LIN {X 0.308,Y -584.908,Z 581.186,A 0.000,B 0.000,C 90.000,E1 69.390} C_DIS
LIN {X -0.011,Y -580.136,Z 581.182,A 0.000,B 0.000,C 90.000,E1 68.773} C_DIS
LIN {X 0.020,Y -575.905,Z 581.179,A 0.000,B 0.000,C 90.000,E1 68.230} C_DIS
LIN {X 0.232,Y -571.249,Z 581.176,A 0.000,B 0.000,C 90.000,E1 67.667} C_DIS
LIN {X -0.295,Y -566.250,Z 581.173,A 0.000,B 0.000,C 90.000,E1 67.177} C_DIS
LIN {X 0.038,Y -560.798,Z 581.170,A 0.000,B 0.000,C 90.000,E1 66.613} C_DIS
LIN {X 0.100,Y -555.120,Z 581.167,A 0.000,B 0.000,C 90.000,E1 66.102} C_DIS
LIN {X 0.102,Y -550.770,Z 581.165,A 0.000,B 0.000,C 90.000,E1 65.741} C_DIS
LIN {X -0.055,Y -544.510,Z 581.163,A 0.000,B 0.000,C 90.000,E1 65.305} C_DIS
LIN {X 0.138,Y -539.632,Z 581.161,A 0.000,B 0.000,C 90.000,E1 64.973} C_DIS
LIN {X 0.129,Y -532.814,Z 581.159,A 0.000,B 0.000,C 90.000,E1 64.588} C_DIS
LIN {X 0.037,Y -527.787,Z 581.157,A 0.000,B 0.000,C 90.000,E1 64.332} C_DIS
LIN {X -0.007,Y -517.436,Z 581.155,A 0.000,B 0.000,C 90.000,E1 63.845} C_DIS
LIN {X -0.005,Y -503.496,Z 581.151,A 0.000,B 0.000,C 90.000,E1 63.256} C_DIS
LIN {X 0.112,Y -476.240,Z 581.145,A 0.000,B 0.000,C 90.000,E1 62.103} C_DIS
LIN {X 0.005,Y -460.881,Z 581.141,A 0.000,B 0.000,C 90.000,E1 61.435} C_DIS
LIN {X 0.181,Y -453.443,Z 581.139,A 0.000,B 0.000,C 90.000,E1 61.051} C_DIS
LIN {X 0.140,Y -453.425,Z 581.139,A 0.000,B 0.000,C 90.000,E1 61.051} C_DIS
LIN {X 0.180,Y -444.954,Z 581.117,A 0.000,B 0.000,C 90.000,E1 57.041} C_DIS
LIN {X -0.068,Y -443.758,Z 581.113,A 0.000,B 0.000,C 90.000,E1 56.421} C_DIS
LIN {X 0.017,Y -435.296,Z 581.093,A 0.000,B 0.000,C 90.000,E1 52.798} C_DIS
LIN {X 0.096,Y -437.237,Z 581.082,A 0.000,B 0.000,C 90.000,E1 50.803} C_DIS
LIN {X -0.065,Y -438.870,Z 581.073,A 0.000,B 0.000,C 90.000,E1 49.175} C_DIS
LIN {X -0.242,Y -440.515,Z 581.064,A 0.000,B 0.000,C 90.000,E1 47.553} C_DIS
LIN {X -0.085,Y -442.174,Z 581.055,A 0.000,B 0.000,C 90.000,E1 45.891} C_DIS
LIN {X -0.210,Y -443.668,Z 581.046,A 0.000,B 0.000,C 90.000,E1 44.271} C_DIS
LIN {X 0.049,Y -444.363,Z 581.040,A 0.000,B 0.000,C 90.000,E1 43.257} C_DIS
LIN {X -0.030,Y -445.165,Z 581.033,A 0.000,B 0.000,C 90.000,E1 41.962} C_DIS
LIN {X 0.265,Y -445.814,Z 581.026,A 0.000,B 0.000,C 90.000,E1 40.620} C_DIS
LIN {X -0.051,Y -446.373,Z 581.019,A 0.000,B 0.000,C 90.000,E1 39.358} C_DIS
LIN {X -0.036,Y -446.814,Z 581.010,A 0.000,B 0.000,C 90.000,E1 37.729} C_DIS
LIN {X 0.006,Y -446.976,Z 581.002,A 0.000,B 0.000,C 90.000,E1 36.423} C_DIS
LIN {X 0.148,Y -446.984,Z 580.995,A 0.000,B 0.000,C 90.000,E1 35.105} C_DIS
LIN {X -0.077,Y -446.839,Z 580.988,A 0.000,B 0.000,C 90.000,E1 33.833} C_DIS
LIN {X 0.024,Y -446.665,Z 580.975,A 0.000,B 0.000,C 90.000,E1 31.544} C_DIS
LIN {X -0.102,Y -446.477,Z 580.963,A 0.000,B 0.000,C 90.000,E1 29.283} C_DIS
LIN {X -0.067,Y -446.370,Z 580.950,A 0.000,B 0.000,C 90.000,E1 27.001} C_DIS
LIN {X -0.040,Y -446.256,Z 580.937,A 0.000,B 0.000,C 90.000,E1 24.719} C_DIS
LIN {X 0.199,Y -446.365,Z 580.930,A 0.000,B 0.000,C 90.000,E1 23.387} C_DIS
LIN {X 0.144,Y -446.539,Z 580.916,A 0.000,B 0.000,C 90.000,E1 20.791} C_DIS
LIN {X -0.247,Y -446.752,Z 580.907,A 0.000,B 0.000,C 90.000,E1 19.214} C_DIS
LIN {X 0.107,Y -447.188,Z 580.892,A 0.000,B 0.000,C 90.000,E1 16.567} C_DIS
LIN {X 0.052,Y -447.892,Z 580.880,A 0.000,B 0.000,C 90.000,E1 14.300} C_DIS
LIN {X -0.028,Y -448.946,Z 580.865,A 0.000,B 0.000,C 90.000,E1 11.715} C_DIS
LIN {X 0.196,Y -450.403,Z 580.851,A 0.000,B 0.000,C 90.000,E1 9.095} C_DIS
LIN {X 0.187,Y -451.893,Z 580.838,A 0.000,B 0.000,C 90.000,E1 6.834} C_DIS
LIN {X -0.185,Y -454.022,Z 580.824,A 0.000,B 0.000,C 90.000,E1 4.302} C_DIS
LIN {X 0.181,Y -456.138,Z 580.811,A 0.000,B 0.000,C 90.000,E1 2.007} C_DIS
LIN {X -0.091,Y -458.975,Z 580.797,A 0.000,B 0.000,C 90.000,E1 359.484} C_DIS
LIN {X 0.140,Y -462.274,Z 580.783,A 0.000,B 0.000,C 90.000,E1 356.906} C_DIS
LIN {X 0.093,Y -465.005,Z 580.772,A 0.000,B 0.000,C 90.000,E1 355.008} C_DIS
LIN {X -0.081,Y -468.314,Z 580.760,A 0.000,B 0.000,C 90.000,E1 352.818} C_DIS
LIN {X 0.216,Y -469.792,Z 580.755,A 0.000,B 0.000,C 90.000,E1 351.837} C_DIS
LIN {X -0.006,Y -472.711,Z 580.744,A 0.000,B 0.000,C 90.000,E1 349.982} C_DIS
LIN {X -0.148,Y -476.086,Z 580.732,A 0.000,B 0.000,C 90.000,E1 347.813} C_DIS
LIN {X 0.233,Y -480.226,Z 580.718,A 0.000,B 0.000,C 90.000,E1 345.283} C_DIS
LIN {X 0.061,Y -484.710,Z 580.705,A 0.000,B 0.000,C 90.000,E1 342.834} C_DIS
LIN {X 0.141,Y -488.837,Z 580.693,A 0.000,B 0.000,C 90.000,E1 340.678} C_DIS
LIN {X 0.140,Y -492.354,Z 580.683,A 0.000,B 0.000,C 90.000,E1 338.847} C_DIS
LIN {X -0.155,Y -494.607,Z 580.676,A 0.000,B 0.000,C 90.000,E1 337.667} C_DIS
LIN {X 0.039,Y -496.830,Z 580.669,A 0.000,B 0.000,C 90.000,E1 336.433} C_DIS
LIN {X 0.070,Y -499.384,Z 580.661,A 0.000,B 0.000,C 90.000,E1 334.921} C_DIS
LIN {X -0.016,Y -502.330,Z 580.651,A 0.000,B 0.000,C 90.000,E1 333.127} C_DIS
LIN {X 0.137,Y -506.065,Z 580.637,A 0.000,B 0.000,C 90.000,E1 330.717} C_DIS
LIN {X -0.120,Y -509.435,Z 580.626,A 0.000,B 0.000,C 90.000,E1 328.663} C_DIS
LIN {X -0.037,Y -512.889,Z 580.614,A 0.000,B 0.000,C 90.000,E1 326.580} C_DIS
LIN {X -0.079,Y -515.990,Z 580.605,A 0.000,B 0.000,C 90.000,E1 324.815} C_DIS
LIN {X 0.016,Y -518.630,Z 580.596,A 0.000,B 0.000,C 90.000,E1 323.336} C_DIS
LIN {X -0.084,Y -522.965,Z 580.583,A 0.000,B 0.000,C 90.000,E1 321.009} C_DIS
LIN {X 0.114,Y -529.618,Z 580.566,A 0.000,B 0.000,C 90.000,E1 317.796} C_DIS
LIN {X -0.093,Y -533.573,Z 580.558,A 0.000,B 0.000,C 90.000,E1 316.377} C_DIS
LIN {X 0.250,Y -534.789,Z 580.556,A 0.000,B 0.000,C 90.000,E1 316.053} C_DIS
LIN {X 0.019,Y -536.190,Z 580.554,A 0.000,B 0.000,C 90.000,E1 315.648} C_DIS
LIN {X 0.026,Y -537.834,Z 580.552,A 0.000,B 0.000,C 90.000,E1 315.324} C_DIS
LIN {X -0.189,Y -540.578,Z 580.549,A 0.000,B 0.000,C 90.000,E1 314.919} C_DIS
LIN {X 0.043,Y -544.352,Z 580.547,A 0.000,B 0.000,C 90.000,E1 314.433} C_DIS
LIN {X -0.320,Y -548.922,Z 580.544,A 0.000,B 0.000,C 90.000,E1 314.028} C_DIS
LIN {X 0.000,Y -553.189,Z 580.542,A 0.000,B 0.000,C 90.000,E1 313.623} C_DIS
LIN {X 0.089,Y -558.609,Z 580.540,A 0.000,B 0.000,C 90.000,E1 313.176} C_DIS
LIN {X 0.161,Y -572.961,Z 580.534,A 0.000,B 0.000,C 90.000,E1 312.123} C_DIS
LIN {X -0.240,Y -592.219,Z 580.526,A 0.000,B 0.000,C 90.000,E1 310.782} C_DIS
LIN {X -0.096,Y -597.922,Z 580.524,A 0.000,B 0.000,C 90.000,E1 310.334} C_DIS
LIN {X -0.088,Y -604.769,Z 580.521,A 0.000,B 0.000,C 90.000,E1 309.769} C_DIS
LIN {X -0.314,Y -611.213,Z 580.518,A 0.000,B 0.000,C 90.000,E1 309.197} C_DIS
LIN {X 0.067,Y -616.222,Z 580.515,A 0.000,B 0.000,C 90.000,E1 308.669} C_DIS
LIN {X -0.076,Y -620.961,Z 580.512,A 0.000,B 0.000,C 90.000,E1 308.177} C_DIS
LIN {X -0.260,Y -624.426,Z 580.510,A 0.000,B 0.000,C 90.000,E1 307.810} C_DIS
LIN {X -0.030,Y -632.937,Z 580.504,A 0.000,B 0.000,C 90.000,E1 306.790} C_DIS
LIN {X -0.173,Y -636.872,Z 580.502,A 0.000,B 0.000,C 90.000,E1 306.297} C_DIS
LIN {X 0.125,Y -643.552,Z 580.497,A 0.000,B 0.000,C 90.000,E1 305.391} C_DIS
LIN {X 0.042,Y -648.595,Z 580.493,A 0.000,B 0.000,C 90.000,E1 304.659} C_DIS
LIN {X -0.175,Y -650.918,Z 580.491,A 0.000,B 0.000,C 90.000,E1 304.326} C_DIS
LIN {X -0.109,Y -654.518,Z 580.487,A 0.000,B 0.000,C 90.000,E1 303.706} C_DIS
LIN {X -0.015,Y -658.416,Z 580.483,A 0.000,B 0.000,C 90.000,E1 302.959} C_DIS
LIN {X 0.058,Y -661.330,Z 580.480,A 0.000,B 0.000,C 90.000,E1 302.339} C_DIS
LIN {X 0.213,Y -664.599,Z 580.476,A 0.000,B 0.000,C 90.000,E1 301.592} C_DIS
LIN {X 0.119,Y -669.758,Z 580.469,A 0.000,B 0.000,C 90.000,E1 300.384} C_DIS
LIN {X 0.016,Y -672.719,Z 580.465,A 0.000,B 0.000,C 90.000,E1 299.667} C_DIS
LIN {X -0.056,Y -675.468,Z 580.461,A 0.000,B 0.000,C 90.000,E1 298.949} C_DIS
LIN {X -0.100,Y -677.959,Z 580.457,A 0.000,B 0.000,C 90.000,E1 298.231} C_DIS
LIN {X 0.279,Y -681.824,Z 580.450,A 0.000,B 0.000,C 90.000,E1 297.001} C_DIS
LIN {X 0.081,Y -683.228,Z 580.448,A 0.000,B 0.000,C 90.000,E1 296.539} C_DIS
LIN {X -0.201,Y -684.258,Z 580.444,A 0.000,B 0.000,C 90.000,E1 295.848} C_DIS
LIN {X 0.013,Y -683.895,Z 580.442,A 0.000,B 0.000,C 90.000,E1 295.591} C_DIS
LIN {X 0.150,Y -682.857,Z 580.440,A 0.000,B 0.000,C 90.000,E1 295.103} C_DIS
LIN {X -0.363,Y -682.292,Z 580.439,A 0.000,B 0.000,C 90.000,E1 295.027} C_DIS
LIN {X -0.256,Y -681.396,Z 580.438,A 0.000,B 0.000,C 90.000,E1 294.899} C_DIS
LIN {X 0.149,Y -677.002,Z 580.436,A 0.000,B 0.000,C 90.000,E1 294.387} C_DIS
LIN {X 0.244,Y -675.191,Z 580.435,A 0.000,B 0.000,C 90.000,E1 294.259} C_DIS
LIN {X -0.231,Y -669.405,Z 580.433,A 0.000,B 0.000,C 90.000,E1 294.027} C_DIS
LIN {X 0.155,Y -667.577,Z 580.433,A 0.000,B 0.000,C 90.000,E1 293.898} C_DIS
LIN {X 0.000,Y -660.359,Z 580.432,A 0.000,B 0.000,C 90.000,E1 293.695} C_DIS
LIN {X -0.005,Y -658.269,Z 580.431,A 0.000,B 0.000,C 90.000,E1 293.643} C_DIS
LIN {X 0.273,Y -632.150,Z 580.428,A 0.000,B 0.000,C 90.000,E1 293.078} C_DIS
LIN {X -0.006,Y -618.722,Z 580.427,A 0.000,B 0.000,C 90.000,E1 292.770} C_DIS
LIN {X 0.232,Y -598.679,Z 580.423,A 0.000,B 0.000,C 90.000,E1 292.153} C_DIS
LIN {X -0.237,Y -572.595,Z 580.419,A 0.000,B 0.000,C 90.000,E1 291.354} C_DIS
LIN {X 0.149,Y -566.186,Z 580.417,A 0.000,B 0.000,C 90.000,E1 291.046} C_DIS
LIN {X -0.102,Y -562.883,Z 580.416,A 0.000,B 0.000,C 90.000,E1 290.844} C_DIS
LIN {X -0.133,Y -562.840,Z 580.416,A 0.000,B 0.000,C 90.000,E1 290.844} C_DIS
LIN {X -0.190,Y -561.903,Z 580.415,A 0.000,B 0.000,C 90.000,E1 290.663} C_DIS
LIN {X -0.175,Y -561.379,Z 580.412,A 0.000,B 0.000,C 90.000,E1 290.248} C_DIS
LIN {X -0.231,Y -561.567,Z 580.405,A 0.000,B 0.000,C 90.000,E1 288.960} C_DIS
LIN {X -0.279,Y -561.238,Z 580.398,A 0.000,B 0.000,C 90.000,E1 287.583} C_DIS
LIN {X -0.069,Y -560.943,Z 580.393,A 0.000,B 0.000,C 90.000,E1 286.732} C_DIS
LIN {X 0.114,Y -560.513,Z 580.387,A 0.000,B 0.000,C 90.000,E1 285.607} C_DIS
LIN {X -0.101,Y -559.747,Z 580.379,A 0.000,B 0.000,C 90.000,E1 284.245} C_DIS
LIN {X 0.212,Y -558.948,Z 580.371,A 0.000,B 0.000,C 90.000,E1 282.827} C_DIS
LIN {X -0.020,Y -558.032,Z 580.362,A 0.000,B 0.000,C 90.000,E1 281.186} C_DIS
LIN {X 0.173,Y -557.035,Z 580.353,A 0.000,B 0.000,C 90.000,E1 279.500} C_DIS
LIN {X -0.158,Y -556.088,Z 580.342,A 0.000,B 0.000,C 90.000,E1 277.587} C_DIS
LIN {X -0.217,Y -555.447,Z 580.334,A 0.000,B 0.000,C 90.000,E1 276.201} C_DIS
LIN {X 0.007,Y -554.575,Z 580.320,A 0.000,B 0.000,C 90.000,E1 273.669} C_DIS
LIN {X -0.014,Y -554.033,Z 580.310,A 0.000,B 0.000,C 90.000,E1 271.718} C_DIS
LIN {X -0.149,Y -553.451,Z 580.300,A 0.000,B 0.000,C 90.000,E1 270.057} C_DIS
LIN {X 0.189,Y -552.885,Z 580.293,A 0.000,B 0.000,C 90.000,E1 268.625} C_DIS
LIN {X 0.129,Y -552.074,Z 580.282,A 0.000,B 0.000,C 90.000,E1 266.674} C_DIS
LIN {X -0.101,Y -551.405,Z 580.274,A 0.000,B 0.000,C 90.000,E1 265.298} C_DIS
LIN {X -0.251,Y -550.616,Z 580.266,A 0.000,B 0.000,C 90.000,E1 263.913} C_DIS
LIN {X 0.037,Y -549.903,Z 580.260,A 0.000,B 0.000,C 90.000,E1 262.761} C_DIS
LIN {X 0.277,Y -549.162,Z 580.255,A 0.000,B 0.000,C 90.000,E1 261.894} C_DIS
LIN {X 0.171,Y -547.801,Z 580.247,A 0.000,B 0.000,C 90.000,E1 260.500} C_DIS
LIN {X -0.109,Y -545.300,Z 580.233,A 0.000,B 0.000,C 90.000,E1 257.993} C_DIS
LIN {X 0.028,Y -543.540,Z 580.224,A 0.000,B 0.000,C 90.000,E1 256.284} C_DIS
LIN {X 0.123,Y -541.724,Z 580.214,A 0.000,B 0.000,C 90.000,E1 254.574} C_DIS
LIN {X 0.028,Y -540.537,Z 580.208,A 0.000,B 0.000,C 90.000,E1 253.449} C_DIS
LIN {X 0.067,Y -539.198,Z 580.202,A 0.000,B 0.000,C 90.000,E1 252.308} C_DIS
LIN {X 0.085,Y -537.687,Z 580.195,A 0.000,B 0.000,C 90.000,E1 251.167} C_DIS
LIN {X -0.039,Y -535.497,Z 580.188,A 0.000,B 0.000,C 90.000,E1 249.752} C_DIS
LIN {X 0.103,Y -533.530,Z 580.181,A 0.000,B 0.000,C 90.000,E1 248.592} C_DIS
LIN {X 0.214,Y -531.881,Z 580.176,A 0.000,B 0.000,C 90.000,E1 247.720} C_DIS
LIN {X -0.011,Y -528.945,Z 580.168,A 0.000,B 0.000,C 90.000,E1 246.305} C_DIS
LIN {X 0.133,Y -525.899,Z 580.160,A 0.000,B 0.000,C 90.000,E1 244.845} C_DIS
LIN {X 0.224,Y -522.723,Z 580.152,A 0.000,B 0.000,C 90.000,E1 243.384} C_DIS
LIN {X 0.111,Y -520.028,Z 580.146,A 0.000,B 0.000,C 90.000,E1 242.231} C_DIS
LIN {X 0.201,Y -517.136,Z 580.139,A 0.000,B 0.000,C 90.000,E1 241.051} C_DIS
LIN {X -0.111,Y -514.849,Z 580.134,A 0.000,B 0.000,C 90.000,E1 240.205} C_DIS
LIN {X 0.161,Y -511.634,Z 580.128,A 0.000,B 0.000,C 90.000,E1 238.997} C_DIS
LIN {X 0.014,Y -507.672,Z 580.120,A 0.000,B 0.000,C 90.000,E1 237.533} C_DIS
LIN {X 0.132,Y -505.254,Z 580.115,A 0.000,B 0.000,C 90.000,E1 236.628} C_DIS
LIN {X -0.284,Y -501.072,Z 580.106,A 0.000,B 0.000,C 90.000,E1 235.182} C_DIS
LIN {X 0.070,Y -491.975,Z 580.088,A 0.000,B 0.000,C 90.000,E1 231.823} C_DIS
LIN {X 0.100,Y -485.568,Z 580.074,A 0.000,B 0.000,C 90.000,E1 229.380} C_DIS
LIN {X -0.122,Y -479.269,Z 580.061,A 0.000,B 0.000,C 90.000,E1 226.944} C_DIS
LIN {X -0.107,Y -474.704,Z 580.050,A 0.000,B 0.000,C 90.000,E1 225.081} C_DIS
LIN {X 0.061,Y -471.030,Z 580.042,A 0.000,B 0.000,C 90.000,E1 223.500} C_DIS
LIN {X 0.227,Y -466.705,Z 580.031,A 0.000,B 0.000,C 90.000,E1 221.595} C_DIS
LIN {X 0.063,Y -461.888,Z 580.019,A 0.000,B 0.000,C 90.000,E1 219.402} C_DIS
LIN {X -0.183,Y -457.842,Z 580.008,A 0.000,B 0.000,C 90.000,E1 217.523} C_DIS
LIN {X 0.029,Y -455.160,Z 580.001,A 0.000,B 0.000,C 90.000,E1 216.217} C_DIS
LIN {X 0.102,Y -451.223,Z 579.991,A 0.000,B 0.000,C 90.000,E1 214.278} C_DIS
LIN {X 0.088,Y -447.488,Z 579.980,A 0.000,B 0.000,C 90.000,E1 212.339} C_DIS
LIN {X -0.051,Y -443.386,Z 579.967,A 0.000,B 0.000,C 90.000,E1 210.079} C_DIS
LIN {X 0.042,Y -439.856,Z 579.956,A 0.000,B 0.000,C 90.000,E1 208.103} C_DIS
LIN {X -0.190,Y -436.993,Z 579.947,A 0.000,B 0.000,C 90.000,E1 206.488} C_DIS
LIN {X 0.127,Y -433.611,Z 579.936,A 0.000,B 0.000,C 90.000,E1 204.463} C_DIS
LIN {X 0.183,Y -430.314,Z 579.925,A 0.000,B 0.000,C 90.000,E1 202.461} C_DIS
LIN {X -0.008,Y -427.234,Z 579.914,A 0.000,B 0.000,C 90.000,E1 200.482} C_DIS
LIN {X -0.029,Y -424.300,Z 579.903,A 0.000,B 0.000,C 90.000,E1 198.471} C_DIS
LIN {X 0.019,Y -421.538,Z 579.891,A 0.000,B 0.000,C 90.000,E1 196.441} C_DIS
LIN {X -0.160,Y -419.418,Z 579.882,A 0.000,B 0.000,C 90.000,E1 194.773} C_DIS
LIN {X -0.082,Y -417.143,Z 579.873,A 0.000,B 0.000,C 90.000,E1 193.063} C_DIS
LIN {X 0.117,Y -412.756,Z 579.855,A 0.000,B 0.000,C 90.000,E1 189.962} C_DIS
LIN {X -0.078,Y -409.511,Z 579.840,A 0.000,B 0.000,C 90.000,E1 187.239} C_DIS
LIN {X -0.053,Y -407.085,Z 579.829,A 0.000,B 0.000,C 90.000,E1 185.163} C_DIS
LIN {X 0.132,Y -403.146,Z 579.807,A 0.000,B 0.000,C 90.000,E1 181.318} C_DIS
LIN {X -0.164,Y -401.108,Z 579.792,A 0.000,B 0.000,C 90.000,E1 178.568} C_DIS
LIN {X -0.157,Y -399.309,Z 579.773,A 0.000,B 0.000,C 90.000,E1 175.065} C_DIS
LIN {X -0.033,Y -398.643,Z 579.759,A 0.000,B 0.000,C 90.000,E1 172.591} C_DIS
LIN {X 0.181,Y -398.286,Z 579.741,A 0.000,B 0.000,C 90.000,E1 169.398} C_DIS
LIN {X -0.180,Y -398.631,Z 579.722,A 0.000,B 0.000,C 90.000,E1 165.936} C_DIS
LIN {X 0.023,Y -399.249,Z 579.708,A 0.000,B 0.000,C 90.000,E1 163.449} C_DIS
LIN {X -0.083,Y -400.233,Z 579.693,A 0.000,B 0.000,C 90.000,E1 160.659} C_DIS
LIN {X 0.048,Y -401.182,Z 579.681,A 0.000,B 0.000,C 90.000,E1 158.539} C_DIS
LIN {X 0.061,Y -402.511,Z 579.665,A 0.000,B 0.000,C 90.000,E1 155.741} C_DIS
LIN {X 0.154,Y -403.230,Z 579.658,A 0.000,B 0.000,C 90.000,E1 154.332} C_DIS
LIN {X -0.023,Y -404.157,Z 579.648,A 0.000,B 0.000,C 90.000,E1 152.615} C_DIS
LIN {X -0.067,Y -404.840,Z 579.640,A 0.000,B 0.000,C 90.000,E1 151.229} C_DIS
LIN {X 0.165,Y -405.618,Z 579.630,A 0.000,B 0.000,C 90.000,E1 149.459} C_DIS
LIN {X 0.142,Y -406.155,Z 579.623,A 0.000,B 0.000,C 90.000,E1 148.074} C_DIS
LIN {X 0.034,Y -406.709,Z 579.611,A 0.000,B 0.000,C 90.000,E1 146.008} C_DIS
LIN {X 0.031,Y -407.099,Z 579.602,A 0.000,B 0.000,C 90.000,E1 144.276} C_DIS
LIN {X -0.060,Y -407.438,Z 579.592,A 0.000,B 0.000,C 90.000,E1 142.557} C_DIS
LIN {X 0.105,Y -407.734,Z 579.582,A 0.000,B 0.000,C 90.000,E1 140.803} C_DIS
LIN {X -0.203,Y -408.076,Z 579.571,A 0.000,B 0.000,C 90.000,E1 138.771} C_DIS
LIN {X -0.226,Y -408.318,Z 579.563,A 0.000,B 0.000,C 90.000,E1 137.391} C_DIS
LIN {X -0.005,Y -408.510,Z 579.548,A 0.000,B 0.000,C 90.000,E1 134.595} C_DIS
LIN {X 0.105,Y -408.746,Z 579.538,A 0.000,B 0.000,C 90.000,E1 132.852} C_DIS
LIN {X -0.061,Y -408.923,Z 579.529,A 0.000,B 0.000,C 90.000,E1 131.148} C_DIS
LIN {X -0.075,Y -408.865,Z 579.521,A 0.000,B 0.000,C 90.000,E1 129.769} C_DIS
LIN {X -0.027,Y -408.644,Z 579.513,A 0.000,B 0.000,C 90.000,E1 128.338} C_DIS
LIN {X 0.019,Y -415.544,Z 579.500,A 0.000,B 0.000,C 90.000,E1 125.964} C_DIS
LIN {X 0.103,Y -425.936,Z 579.477,A 0.000,B 0.000,C 90.000,E1 121.878} C_DIS
LIN {X 0.056,Y -430.944,Z 579.468,A 0.000,B 0.000,C 90.000,E1 120.207} C_DIS
LIN {X 0.025,Y -432.452,Z 579.464,A 0.000,B 0.000,C 90.000,E1 119.539} C_DIS
LIN {X -0.014,Y -432.527,Z 579.464,A 0.000,B 0.000,C 90.000,E1 119.539} C_DIS
LIN {X 0.020,Y -450.020,Z 579.460,A 0.000,B 0.000,C 90.000,E1 118.743} C_DIS
LIN {X 0.056,Y -470.512,Z 579.454,A 0.000,B 0.000,C 90.000,E1 117.769} C_DIS
LIN {X -0.135,Y -482.285,Z 579.451,A 0.000,B 0.000,C 90.000,E1 117.206} C_DIS
LIN {X -0.248,Y -488.933,Z 579.449,A 0.000,B 0.000,C 90.000,E1 116.873} C_DIS
LIN {X 0.252,Y -497.099,Z 579.447,A 0.000,B 0.000,C 90.000,E1 116.360} C_DIS
LIN {X 0.075,Y -508.510,Z 579.443,A 0.000,B 0.000,C 90.000,E1 115.720} C_DIS
LIN {X 0.263,Y -516.409,Z 579.440,A 0.000,B 0.000,C 90.000,E1 115.207} C_DIS
LIN {X 0.035,Y -522.640,Z 579.438,A 0.000,B 0.000,C 90.000,E1 114.823} C_DIS
LIN {X -0.331,Y -530.462,Z 579.435,A 0.000,B 0.000,C 90.000,E1 114.335} C_DIS
LIN {X -0.211,Y -537.899,Z 579.432,A 0.000,B 0.000,C 90.000,E1 113.770} C_DIS
LIN {X 0.206,Y -542.356,Z 579.430,A 0.000,B 0.000,C 90.000,E1 113.387} C_DIS
LIN {X -0.102,Y -548.016,Z 579.427,A 0.000,B 0.000,C 90.000,E1 112.950} C_DIS
LIN {X -0.113,Y -552.213,Z 579.425,A 0.000,B 0.000,C 90.000,E1 112.589} C_DIS
LIN {X -0.037,Y -557.502,Z 579.423,A 0.000,B 0.000,C 90.000,E1 112.078} C_DIS
LIN {X 0.017,Y -562.507,Z 579.420,A 0.000,B 0.000,C 90.000,E1 111.535} C_DIS
LIN {X 0.232,Y -565.857,Z 579.417,A 0.000,B 0.000,C 90.000,E1 111.099} C_DIS
LIN {X 0.130,Y -567.039,Z 579.417,A 0.000,B 0.000,C 90.000,E1 110.972} C_DIS
LIN {X 0.169,Y -569.961,Z 579.414,A 0.000,B 0.000,C 90.000,E1 110.556} C_DIS
LIN {X -0.020,Y -571.984,Z 579.413,A 0.000,B 0.000,C 90.000,E1 110.301} C_DIS
LIN {X 0.047,Y -574.436,Z 579.411,A 0.000,B 0.000,C 90.000,E1 109.885} C_DIS
LIN {X -0.311,Y -577.683,Z 579.408,A 0.000,B 0.000,C 90.000,E1 109.396} C_DIS
LIN {X -0.102,Y -580.786,Z 579.405,A 0.000,B 0.000,C 90.000,E1 108.833} C_DIS
LIN {X 0.154,Y -584.940,Z 579.400,A 0.000,B 0.000,C 90.000,E1 108.000} C_DIS
LIN {X -0.097,Y -588.746,Z 579.396,A 0.000,B 0.000,C 90.000,E1 107.221} C_DIS
LIN {X -0.312,Y -592.321,Z 579.391,A 0.000,B 0.000,C 90.000,E1 106.441} C_DIS
LIN {X -0.226,Y -596.739,Z 579.385,A 0.000,B 0.000,C 90.000,E1 105.371} C_DIS
LIN {X -0.082,Y -598.762,Z 579.382,A 0.000,B 0.000,C 90.000,E1 104.828} C_DIS
LIN {X -0.058,Y -602.657,Z 579.377,A 0.000,B 0.000,C 90.000,E1 103.772} C_DIS
LIN {X -0.169,Y -609.216,Z 579.366,A 0.000,B 0.000,C 90.000,E1 101.951} C_DIS
LIN {X 0.108,Y -614.874,Z 579.358,A 0.000,B 0.000,C 90.000,E1 100.366} C_DIS
LIN {X 0.242,Y -618.538,Z 579.352,A 0.000,B 0.000,C 90.000,E1 99.321} C_DIS
LIN {X -0.280,Y -622.050,Z 579.346,A 0.000,B 0.000,C 90.000,E1 98.341} C_DIS
LIN {X -0.049,Y -625.451,Z 579.341,A 0.000,B 0.000,C 90.000,E1 97.296} C_DIS
LIN {X 0.146,Y -628.687,Z 579.335,A 0.000,B 0.000,C 90.000,E1 96.258} C_DIS
LIN {X -0.022,Y -630.938,Z 579.331,A 0.000,B 0.000,C 90.000,E1 95.511} C_DIS
LIN {X -0.112,Y -633.026,Z 579.326,A 0.000,B 0.000,C 90.000,E1 94.759} C_DIS
LIN {X 0.129,Y -635.367,Z 579.321,A 0.000,B 0.000,C 90.000,E1 93.726} C_DIS
LIN {X 0.024,Y -636.872,Z 579.317,A 0.000,B 0.000,C 90.000,E1 92.980} C_DIS
LIN {X -0.096,Y -638.283,Z 579.312,A 0.000,B 0.000,C 90.000,E1 92.236} C_DIS
LIN {X -0.178,Y -639.470,Z 579.308,A 0.000,B 0.000,C 90.000,E1 91.489} C_DIS
LIN {X 0.133,Y -640.660,Z 579.303,A 0.000,B 0.000,C 90.000,E1 90.458} C_DIS
LIN {X 0.059,Y -641.301,Z 579.298,A 0.000,B 0.000,C 90.000,E1 89.714} C_DIS
LIN {X -0.009,Y -641.704,Z 579.294,A 0.000,B 0.000,C 90.000,E1 88.969} C_DIS
LIN {X -0.079,Y -641.787,Z 579.290,A 0.000,B 0.000,C 90.000,E1 88.224} C_DIS
LIN {X 0.278,Y -641.521,Z 579.285,A 0.000,B 0.000,C 90.000,E1 87.192} C_DIS
LIN {X 0.234,Y -641.094,Z 579.280,A 0.000,B 0.000,C 90.000,E1 86.445} C_DIS
LIN {X -0.056,Y -640.223,Z 579.275,A 0.000,B 0.000,C 90.000,E1 85.469} C_DIS
LIN {X 0.333,Y -639.053,Z 579.269,A 0.000,B 0.000,C 90.000,E1 84.432} C_DIS
LIN {X -0.111,Y -638.402,Z 579.266,A 0.000,B 0.000,C 90.000,E1 83.970} C_DIS
LIN {X 0.259,Y -636.795,Z 579.261,A 0.000,B 0.000,C 90.000,E1 82.932} C_DIS
LIN {X 0.160,Y -635.277,Z 579.257,A 0.000,B 0.000,C 90.000,E1 82.186} C_DIS
LIN {X -0.062,Y -633.032,Z 579.251,A 0.000,B 0.000,C 90.000,E1 81.197} C_DIS
LIN {X -0.112,Y -631.199,Z 579.247,A 0.000,B 0.000,C 90.000,E1 80.443} C_DIS
LIN {X 0.236,Y -628.482,Z 579.241,A 0.000,B 0.000,C 90.000,E1 79.398} C_DIS
LIN {X -0.073,Y -625.599,Z 579.236,A 0.000,B 0.000,C 90.000,E1 78.409} C_DIS
LIN {X -0.295,Y -622.502,Z 579.230,A 0.000,B 0.000,C 90.000,E1 77.409} C_DIS
LIN {X 0.270,Y -619.915,Z 579.226,A 0.000,B 0.000,C 90.000,E1 76.589} C_DIS
LIN {X 0.201,Y -617.142,Z 579.221,A 0.000,B 0.000,C 90.000,E1 75.825} C_DIS
LIN {X 0.259,Y -614.243,Z 579.217,A 0.000,B 0.000,C 90.000,E1 75.046} C_DIS
LIN {X 0.128,Y -611.065,Z 579.213,A 0.000,B 0.000,C 90.000,E1 74.283} C_DIS
LIN {X 0.130,Y -607.605,Z 579.208,A 0.000,B 0.000,C 90.000,E1 73.504} C_DIS
LIN {X 0.050,Y -603.190,Z 579.203,A 0.000,B 0.000,C 90.000,E1 72.598} C_DIS
LIN {X -0.073,Y -597.683,Z 579.198,A 0.000,B 0.000,C 90.000,E1 71.583} C_DIS
LIN {X 0.101,Y -593.982,Z 579.194,A 0.000,B 0.000,C 90.000,E1 70.913} C_DIS
LIN {X 0.221,Y -588.281,Z 579.189,A 0.000,B 0.000,C 90.000,E1 70.007} C_DIS
LIN {X -0.236,Y -584.628,Z 579.186,A 0.000,B 0.000,C 90.000,E1 69.518} C_DIS
LIN {X 0.037,Y -580.649,Z 579.183,A 0.000,B 0.000,C 90.000,E1 68.954} C_DIS
LIN {X -0.131,Y -575.504,Z 579.180,A 0.000,B 0.000,C 90.000,E1 68.337} C_DIS
LIN {X 0.265,Y -571.069,Z 579.177,A 0.000,B 0.000,C 90.000,E1 67.794} C_DIS
LIN {X 0.104,Y -565.017,Z 579.173,A 0.000,B 0.000,C 90.000,E1 67.177} C_DIS
LIN {X 0.309,Y -561.269,Z 579.171,A 0.000,B 0.000,C 90.000,E1 66.794} C_DIS
LIN {X 0.031,Y -556.038,Z 579.169,A 0.000,B 0.000,C 90.000,E1 66.357} C_DIS
LIN {X -0.113,Y -550.476,Z 579.166,A 0.000,B 0.000,C 90.000,E1 65.921} C_DIS
LIN {X -0.272,Y -544.106,Z 579.164,A 0.000,B 0.000,C 90.000,E1 65.485} C_DIS
LIN {X -0.084,Y -539.070,Z 579.162,A 0.000,B 0.000,C 90.000,E1 65.153} C_DIS
LIN {X -0.184,Y -532.318,Z 579.160,A 0.000,B 0.000,C 90.000,E1 64.793} C_DIS
LIN {X -0.242,Y -527.296,Z 579.158,A 0.000,B 0.000,C 90.000,E1 64.537} C_DIS
LIN {X -0.051,Y -516.811,Z 579.156,A 0.000,B 0.000,C 90.000,E1 64.024} C_DIS
LIN {X -0.108,Y -501.135,Z 579.152,A 0.000,B 0.000,C 90.000,E1 63.384} C_DIS
LIN {X 0.003,Y -471.916,Z 579.145,A 0.000,B 0.000,C 90.000,E1 62.153} C_DIS
LIN {X -0.103,Y -458.508,Z 579.142,A 0.000,B 0.000,C 90.000,E1 61.563} C_DIS
LIN {X 0.267,Y -454.174,Z 579.141,A 0.000,B 0.000,C 90.000,E1 61.307} C_DIS
LIN {X 0.226,Y -454.082,Z 579.141,A 0.000,B 0.000,C 90.000,E1 61.307} C_DIS
LIN {X 0.113,Y -445.458,Z 579.119,A 0.000,B 0.000,C 90.000,E1 57.327} C_DIS
LIN {X -0.076,Y -443.629,Z 579.113,A 0.000,B 0.000,C 90.000,E1 56.373} C_DIS
LIN {X 0.064,Y -435.664,Z 579.094,A 0.000,B 0.000,C 90.000,E1 52.970} C_DIS
LIN {X -0.269,Y -437.926,Z 579.082,A 0.000,B 0.000,C 90.000,E1 50.803} C_DIS
LIN {X -0.131,Y -439.606,Z 579.073,A 0.000,B 0.000,C 90.000,E1 49.138} C_DIS
LIN {X 0.041,Y -441.307,Z 579.064,A 0.000,B 0.000,C 90.000,E1 47.472} C_DIS
LIN {X 0.216,Y -442.997,Z 579.055,A 0.000,B 0.000,C 90.000,E1 45.810} C_DIS
LIN {X 0.127,Y -444.205,Z 579.047,A 0.000,B 0.000,C 90.000,E1 44.514} C_DIS
LIN {X 0.071,Y -444.992,Z 579.042,A 0.000,B 0.000,C 90.000,E1 43.542} C_DIS
LIN {X 0.029,Y -445.822,Z 579.035,A 0.000,B 0.000,C 90.000,E1 42.243} C_DIS
LIN {X 0.006,Y -446.496,Z 579.028,A 0.000,B 0.000,C 90.000,E1 40.943} C_DIS
LIN {X -0.011,Y -447.051,Z 579.020,A 0.000,B 0.000,C 90.000,E1 39.644} C_DIS
LIN {X 0.040,Y -447.436,Z 579.013,A 0.000,B 0.000,C 90.000,E1 38.338} C_DIS
LIN {X 0.100,Y -447.659,Z 579.006,A 0.000,B 0.000,C 90.000,E1 37.030} C_DIS
LIN {X 0.157,Y -447.733,Z 578.999,A 0.000,B 0.000,C 90.000,E1 35.724} C_DIS
LIN {X 0.011,Y -447.546,Z 578.990,A 0.000,B 0.000,C 90.000,E1 34.119} C_DIS
LIN {X -0.245,Y -447.280,Z 578.977,A 0.000,B 0.000,C 90.000,E1 31.878} C_DIS
LIN {X 0.185,Y -447.085,Z 578.966,A 0.000,B 0.000,C 90.000,E1 29.873} C_DIS
LIN {X -0.146,Y -446.992,Z 578.959,A 0.000,B 0.000,C 90.000,E1 28.615} C_DIS
LIN {X -0.233,Y -446.874,Z 578.950,A 0.000,B 0.000,C 90.000,E1 27.001} C_DIS
LIN {X -0.060,Y -446.713,Z 578.939,A 0.000,B 0.000,C 90.000,E1 25.027} C_DIS
LIN {X 0.054,Y -446.776,Z 578.930,A 0.000,B 0.000,C 90.000,E1 23.387} C_DIS
LIN {X 0.141,Y -446.925,Z 578.917,A 0.000,B 0.000,C 90.000,E1 21.099} C_DIS
LIN {X 0.196,Y -447.102,Z 578.907,A 0.000,B 0.000,C 90.000,E1 19.141} C_DIS
LIN {X -0.007,Y -447.486,Z 578.892,A 0.000,B 0.000,C 90.000,E1 16.567} C_DIS
LIN {X -0.054,Y -448.174,Z 578.879,A 0.000,B 0.000,C 90.000,E1 14.300} C_DIS
LIN {X -0.126,Y -449.216,Z 578.865,A 0.000,B 0.000,C 90.000,E1 11.715} C_DIS
LIN {X -0.142,Y -450.845,Z 578.849,A 0.000,B 0.000,C 90.000,E1 8.803} C_DIS
LIN {X -0.147,Y -452.348,Z 578.836,A 0.000,B 0.000,C 90.000,E1 6.543} C_DIS
LIN {X -0.064,Y -454.495,Z 578.822,A 0.000,B 0.000,C 90.000,E1 3.955} C_DIS
LIN {X -0.153,Y -456.621,Z 578.810,A 0.000,B 0.000,C 90.000,E1 1.718} C_DIS
LIN {X -0.090,Y -459.111,Z 578.797,A 0.000,B 0.000,C 90.000,E1 359.484} C_DIS
LIN {X 0.144,Y -462.399,Z 578.783,A 0.000,B 0.000,C 90.000,E1 356.906} C_DIS
LIN {X 0.101,Y -465.118,Z 578.772,A 0.000,B 0.000,C 90.000,E1 355.008} C_DIS
LIN {X -0.071,Y -468.411,Z 578.760,A 0.000,B 0.000,C 90.000,E1 352.818} C_DIS
LIN {X 0.228,Y -469.885,Z 578.755,A 0.000,B 0.000,C 90.000,E1 351.837} C_DIS
LIN {X 0.008,Y -472.795,Z 578.744,A 0.000,B 0.000,C 90.000,E1 349.982} C_DIS
LIN {X -0.131,Y -476.160,Z 578.732,A 0.000,B 0.000,C 90.000,E1 347.813} C_DIS
LIN {X 0.101,Y -480.818,Z 578.717,A 0.000,B 0.000,C 90.000,E1 344.991} C_DIS
LIN {X -0.063,Y -484.724,Z 578.705,A 0.000,B 0.000,C 90.000,E1 342.851} C_DIS
LIN {X 0.161,Y -488.870,Z 578.693,A 0.000,B 0.000,C 90.000,E1 340.678} C_DIS
LIN {X 0.161,Y -492.383,Z 578.683,A 0.000,B 0.000,C 90.000,E1 338.847} C_DIS
LIN {X -0.134,Y -494.669,Z 578.676,A 0.000,B 0.000,C 90.000,E1 337.667} C_DIS
LIN {X 0.114,Y -497.400,Z 578.667,A 0.000,B 0.000,C 90.000,E1 336.125} C_DIS
LIN {X -0.299,Y -499.940,Z 578.659,A 0.000,B 0.000,C 90.000,E1 334.665} C_DIS
LIN {X 0.009,Y -502.421,Z 578.651,A 0.000,B 0.000,C 90.000,E1 333.127} C_DIS
LIN {X -0.148,Y -505.683,Z 578.639,A 0.000,B 0.000,C 90.000,E1 331.051} C_DIS
LIN {X -0.089,Y -509.555,Z 578.626,A 0.000,B 0.000,C 90.000,E1 328.663} C_DIS
LIN {X -0.001,Y -513.014,Z 578.614,A 0.000,B 0.000,C 90.000,E1 326.580} C_DIS
LIN {X -0.041,Y -516.104,Z 578.605,A 0.000,B 0.000,C 90.000,E1 324.815} C_DIS
LIN {X 0.057,Y -518.741,Z 578.596,A 0.000,B 0.000,C 90.000,E1 323.336} C_DIS
LIN {X -0.085,Y -523.629,Z 578.582,A 0.000,B 0.000,C 90.000,E1 320.723} C_DIS
LIN {X 0.066,Y -531.042,Z 578.563,A 0.000,B 0.000,C 90.000,E1 317.229} C_DIS
LIN {X -0.046,Y -533.355,Z 578.558,A 0.000,B 0.000,C 90.000,E1 316.377} C_DIS
LIN {X 0.038,Y -536.662,Z 578.552,A 0.000,B 0.000,C 90.000,E1 315.364} C_DIS
LIN {X -0.167,Y -537.381,Z 578.551,A 0.000,B 0.000,C 90.000,E1 315.243} C_DIS
LIN {X -0.073,Y -539.949,Z 578.549,A 0.000,B 0.000,C 90.000,E1 314.798} C_DIS
LIN {X -0.270,Y -540.604,Z 578.548,A 0.000,B 0.000,C 90.000,E1 314.676} C_DIS
LIN {X 0.294,Y -543.707,Z 578.546,A 0.000,B 0.000,C 90.000,E1 314.190} C_DIS
LIN {X -0.090,Y -546.253,Z 578.544,A 0.000,B 0.000,C 90.000,E1 313.947} C_DIS
LIN {X 0.130,Y -552.623,Z 578.541,A 0.000,B 0.000,C 90.000,E1 313.338} C_DIS
LIN {X 0.077,Y -557.032,Z 578.539,A 0.000,B 0.000,C 90.000,E1 312.975} C_DIS
LIN {X -0.113,Y -571.603,Z 578.533,A 0.000,B 0.000,C 90.000,E1 311.919} C_DIS
LIN {X -0.168,Y -590.973,Z 578.525,A 0.000,B 0.000,C 90.000,E1 310.539} C_DIS
LIN {X 0.048,Y -596.651,Z 578.523,A 0.000,B 0.000,C 90.000,E1 310.092} C_DIS
LIN {X 0.079,Y -602.162,Z 578.520,A 0.000,B 0.000,C 90.000,E1 309.644} C_DIS
LIN {X 0.324,Y -606.178,Z 578.518,A 0.000,B 0.000,C 90.000,E1 309.277} C_DIS
LIN {X 0.007,Y -611.266,Z 578.516,A 0.000,B 0.000,C 90.000,E1 308.830} C_DIS
LIN {X -0.016,Y -615.024,Z 578.514,A 0.000,B 0.000,C 90.000,E1 308.463} C_DIS
LIN {X -0.156,Y -619.793,Z 578.511,A 0.000,B 0.000,C 90.000,E1 307.971} C_DIS
LIN {X 0.344,Y -626.720,Z 578.507,A 0.000,B 0.000,C 90.000,E1 307.156} C_DIS
LIN {X -0.353,Y -632.016,Z 578.503,A 0.000,B 0.000,C 90.000,E1 306.583} C_DIS
LIN {X -0.090,Y -637.967,Z 578.499,A 0.000,B 0.000,C 90.000,E1 305.804} C_DIS
LIN {X 0.204,Y -643.555,Z 578.495,A 0.000,B 0.000,C 90.000,E1 305.025} C_DIS
LIN {X 0.131,Y -647.050,Z 578.492,A 0.000,B 0.000,C 90.000,E1 304.532} C_DIS
LIN {X 0.115,Y -651.053,Z 578.489,A 0.000,B 0.000,C 90.000,E1 303.913} C_DIS
LIN {X -0.314,Y -653.292,Z 578.486,A 0.000,B 0.000,C 90.000,E1 303.579} C_DIS
LIN {X -0.232,Y -657.219,Z 578.482,A 0.000,B 0.000,C 90.000,E1 302.832} C_DIS
LIN {X -0.222,Y -659.666,Z 578.480,A 0.000,B 0.000,C 90.000,E1 302.339} C_DIS
LIN {X 0.359,Y -661.948,Z 578.477,A 0.000,B 0.000,C 90.000,E1 301.799} C_DIS
LIN {X 0.177,Y -665.134,Z 578.473,A 0.000,B 0.000,C 90.000,E1 301.082} C_DIS
LIN {X 0.099,Y -670.238,Z 578.466,A 0.000,B 0.000,C 90.000,E1 299.873} C_DIS
LIN {X 0.006,Y -673.077,Z 578.462,A 0.000,B 0.000,C 90.000,E1 299.155} C_DIS
LIN {X -0.058,Y -675.691,Z 578.458,A 0.000,B 0.000,C 90.000,E1 298.437} C_DIS
LIN {X -0.316,Y -679.610,Z 578.451,A 0.000,B 0.000,C 90.000,E1 297.257} C_DIS
LIN {X 0.080,Y -681.142,Z 578.449,A 0.000,B 0.000,C 90.000,E1 296.744} C_DIS
LIN {X 0.283,Y -681.751,Z 578.447,A 0.000,B 0.000,C 90.000,E1 296.488} C_DIS
LIN {X 0.082,Y -682.489,Z 578.445,A 0.000,B 0.000,C 90.000,E1 296.027} C_DIS
LIN {X -0.009,Y -682.669,Z 578.443,A 0.000,B 0.000,C 90.000,E1 295.796} C_DIS
LIN {X 0.202,Y -682.419,Z 578.442,A 0.000,B 0.000,C 90.000,E1 295.540} C_DIS
LIN {X -0.205,Y -681.923,Z 578.441,A 0.000,B 0.000,C 90.000,E1 295.335} C_DIS
LIN {X 0.002,Y -681.192,Z 578.439,A 0.000,B 0.000,C 90.000,E1 295.079} C_DIS
LIN {X 0.022,Y -678.656,Z 578.437,A 0.000,B 0.000,C 90.000,E1 294.719} C_DIS
LIN {X 0.220,Y -676.518,Z 578.436,A 0.000,B 0.000,C 90.000,E1 294.463} C_DIS
LIN {X 0.316,Y -675.021,Z 578.435,A 0.000,B 0.000,C 90.000,E1 294.335} C_DIS
LIN {X -0.089,Y -670.716,Z 578.434,A 0.000,B 0.000,C 90.000,E1 294.155} C_DIS
LIN {X -0.123,Y -666.987,Z 578.433,A 0.000,B 0.000,C 90.000,E1 293.951} C_DIS
LIN {X 0.276,Y -662.448,Z 578.432,A 0.000,B 0.000,C 90.000,E1 293.770} C_DIS
LIN {X -0.053,Y -656.828,Z 578.431,A 0.000,B 0.000,C 90.000,E1 293.643} C_DIS
LIN {X 0.005,Y -645.236,Z 578.430,A 0.000,B 0.000,C 90.000,E1 293.387} C_DIS
LIN {X 0.130,Y -631.419,Z 578.428,A 0.000,B 0.000,C 90.000,E1 293.078} C_DIS
LIN {X -0.181,Y -617.849,Z 578.426,A 0.000,B 0.000,C 90.000,E1 292.770} C_DIS
LIN {X 0.232,Y -594.437,Z 578.423,A 0.000,B 0.000,C 90.000,E1 292.025} C_DIS
LIN {X 0.126,Y -573.612,Z 578.419,A 0.000,B 0.000,C 90.000,E1 291.354} C_DIS
LIN {X 0.201,Y -566.446,Z 578.417,A 0.000,B 0.000,C 90.000,E1 291.046} C_DIS
LIN {X -0.125,Y -563.131,Z 578.416,A 0.000,B 0.000,C 90.000,E1 290.844} C_DIS
LIN {X -0.159,Y -563.106,Z 578.416,A 0.000,B 0.000,C 90.000,E1 290.844} C_DIS
LIN {X 0.244,Y -562.230,Z 578.415,A 0.000,B 0.000,C 90.000,E1 290.610} C_DIS
LIN {X -0.266,Y -561.819,Z 578.412,A 0.000,B 0.000,C 90.000,E1 290.248} C_DIS
LIN {X -0.254,Y -561.969,Z 578.405,A 0.000,B 0.000,C 90.000,E1 288.906} C_DIS
LIN {X -0.121,Y -561.641,Z 578.397,A 0.000,B 0.000,C 90.000,E1 287.511} C_DIS
LIN {X -0.027,Y -561.016,Z 578.388,A 0.000,B 0.000,C 90.000,E1 285.843} C_DIS
LIN {X -0.234,Y -560.281,Z 578.380,A 0.000,B 0.000,C 90.000,E1 284.481} C_DIS
LIN {X 0.090,Y -559.478,Z 578.373,A 0.000,B 0.000,C 90.000,E1 283.063} C_DIS
LIN {X 0.015,Y -558.368,Z 578.362,A 0.000,B 0.000,C 90.000,E1 281.130} C_DIS
LIN {X 0.172,Y -557.541,Z 578.354,A 0.000,B 0.000,C 90.000,E1 279.726} C_DIS
LIN {X -0.158,Y -556.554,Z 578.343,A 0.000,B 0.000,C 90.000,E1 277.814} C_DIS
LIN {X -0.214,Y -555.960,Z 578.336,A 0.000,B 0.000,C 90.000,E1 276.429} C_DIS
LIN {X -0.090,Y -555.141,Z 578.323,A 0.000,B 0.000,C 90.000,E1 274.188} C_DIS
LIN {X -0.085,Y -554.561,Z 578.312,A 0.000,B 0.000,C 90.000,E1 272.236} C_DIS
LIN {X -0.194,Y -554.004,Z 578.303,A 0.000,B 0.000,C 90.000,E1 270.573} C_DIS
LIN {X 0.225,Y -553.321,Z 578.294,A 0.000,B 0.000,C 90.000,E1 268.854} C_DIS
LIN {X 0.147,Y -552.505,Z 578.283,A 0.000,B 0.000,C 90.000,E1 266.906} C_DIS
LIN {X -0.040,Y -551.867,Z 578.275,A 0.000,B 0.000,C 90.000,E1 265.527} C_DIS
LIN {X -0.235,Y -551.106,Z 578.267,A 0.000,B 0.000,C 90.000,E1 264.147} C_DIS
LIN {X 0.159,Y -550.202,Z 578.260,A 0.000,B 0.000,C 90.000,E1 262.704} C_DIS
LIN {X -0.143,Y -549.453,Z 578.255,A 0.000,B 0.000,C 90.000,E1 261.894} C_DIS
LIN {X -0.243,Y -548.057,Z 578.247,A 0.000,B 0.000,C 90.000,E1 260.500} C_DIS
LIN {X -0.074,Y -545.847,Z 578.235,A 0.000,B 0.000,C 90.000,E1 258.229} C_DIS
LIN {X -0.143,Y -544.395,Z 578.227,A 0.000,B 0.000,C 90.000,E1 256.825} C_DIS
LIN {X 0.181,Y -542.303,Z 578.216,A 0.000,B 0.000,C 90.000,E1 254.810} C_DIS
LIN {X 0.097,Y -541.090,Z 578.209,A 0.000,B 0.000,C 90.000,E1 253.685} C_DIS
LIN {X -0.314,Y -539.376,Z 578.202,A 0.000,B 0.000,C 90.000,E1 252.308} C_DIS
LIN {X -0.119,Y -537.820,Z 578.195,A 0.000,B 0.000,C 90.000,E1 251.148} C_DIS
LIN {X -0.153,Y -536.519,Z 578.190,A 0.000,B 0.000,C 90.000,E1 250.296} C_DIS
LIN {X 0.009,Y -534.626,Z 578.184,A 0.000,B 0.000,C 90.000,E1 249.135} C_DIS
LIN {X 0.138,Y -532.525,Z 578.178,A 0.000,B 0.000,C 90.000,E1 247.975} C_DIS
LIN {X 0.133,Y -529.600,Z 578.170,A 0.000,B 0.000,C 90.000,E1 246.538} C_DIS
LIN {X 0.075,Y -526.556,Z 578.162,A 0.000,B 0.000,C 90.000,E1 245.101} C_DIS
LIN {X 0.178,Y -523.365,Z 578.154,A 0.000,B 0.000,C 90.000,E1 243.640} C_DIS
LIN {X 0.075,Y -520.698,Z 578.147,A 0.000,B 0.000,C 90.000,E1 242.487} C_DIS
LIN {X 0.176,Y -517.841,Z 578.141,A 0.000,B 0.000,C 90.000,E1 241.307} C_DIS
LIN {X -0.126,Y -515.592,Z 578.136,A 0.000,B 0.000,C 90.000,E1 240.461} C_DIS
LIN {X -0.103,Y -512.357,Z 578.129,A 0.000,B 0.000,C 90.000,E1 239.282} C_DIS
LIN {X -0.067,Y -507.518,Z 578.119,A 0.000,B 0.000,C 90.000,E1 237.502} C_DIS
LIN {X 0.093,Y -504.245,Z 578.113,A 0.000,B 0.000,C 90.000,E1 236.294} C_DIS
LIN {X -0.057,Y -500.014,Z 578.105,A 0.000,B 0.000,C 90.000,E1 234.815} C_DIS
LIN {X 0.102,Y -491.793,Z 578.088,A 0.000,B 0.000,C 90.000,E1 231.778} C_DIS
LIN {X -0.255,Y -485.399,Z 578.074,A 0.000,B 0.000,C 90.000,E1 229.380} C_DIS
LIN {X -0.275,Y -479.872,Z 578.062,A 0.000,B 0.000,C 90.000,E1 227.229} C_DIS
LIN {X 0.102,Y -475.322,Z 578.052,A 0.000,B 0.000,C 90.000,E1 225.324} C_DIS
LIN {X 0.029,Y -470.868,Z 578.042,A 0.000,B 0.000,C 90.000,E1 223.461} C_DIS
LIN {X -0.129,Y -466.548,Z 578.031,A 0.000,B 0.000,C 90.000,E1 221.595} C_DIS
LIN {X 0.064,Y -461.728,Z 578.019,A 0.000,B 0.000,C 90.000,E1 219.358} C_DIS
LIN {X 0.101,Y -457.658,Z 578.008,A 0.000,B 0.000,C 90.000,E1 217.443} C_DIS
LIN {X 0.038,Y -455.003,Z 578.001,A 0.000,B 0.000,C 90.000,E1 216.171} C_DIS
LIN {X -0.002,Y -451.040,Z 577.990,A 0.000,B 0.000,C 90.000,E1 214.246} C_DIS
LIN {X 0.105,Y -447.294,Z 577.979,A 0.000,B 0.000,C 90.000,E1 212.291} C_DIS
LIN {X 0.134,Y -443.748,Z 577.969,A 0.000,B 0.000,C 90.000,E1 210.335} C_DIS
LIN {X 0.137,Y -441.395,Z 577.961,A 0.000,B 0.000,C 90.000,E1 209.027} C_DIS
LIN {X 0.143,Y -438.528,Z 577.952,A 0.000,B 0.000,C 90.000,E1 207.385} C_DIS
LIN {X 0.099,Y -435.101,Z 577.941,A 0.000,B 0.000,C 90.000,E1 205.412} C_DIS
LIN {X -0.031,Y -431.755,Z 577.930,A 0.000,B 0.000,C 90.000,E1 203.439} C_DIS
LIN {X 0.012,Y -428.071,Z 577.917,A 0.000,B 0.000,C 90.000,E1 201.099} C_DIS
LIN {X 0.211,Y -424.654,Z 577.904,A 0.000,B 0.000,C 90.000,E1 198.725} C_DIS
LIN {X 0.050,Y -421.417,Z 577.891,A 0.000,B 0.000,C 90.000,E1 196.386} C_DIS
LIN {X -0.128,Y -419.297,Z 577.882,A 0.000,B 0.000,C 90.000,E1 194.717} C_DIS
LIN {X -0.048,Y -417.036,Z 577.872,A 0.000,B 0.000,C 90.000,E1 193.008} C_DIS
LIN {X 0.110,Y -413.128,Z 577.857,A 0.000,B 0.000,C 90.000,E1 190.254} C_DIS
LIN {X -0.070,Y -409.818,Z 577.842,A 0.000,B 0.000,C 90.000,E1 187.530} C_DIS
LIN {X -0.031,Y -407.450,Z 577.830,A 0.000,B 0.000,C 90.000,E1 185.454} C_DIS
LIN {X -0.090,Y -405.109,Z 577.819,A 0.000,B 0.000,C 90.000,E1 183.383} C_DIS
LIN {X -0.009,Y -401.865,Z 577.797,A 0.000,B 0.000,C 90.000,E1 179.542} C_DIS
LIN {X 0.082,Y -400.133,Z 577.782,A 0.000,B 0.000,C 90.000,E1 176.731} C_DIS
LIN {X 0.092,Y -398.887,Z 577.762,A 0.000,B 0.000,C 90.000,E1 173.223} C_DIS
LIN {X -0.153,Y -398.415,Z 577.743,A 0.000,B 0.000,C 90.000,E1 169.746} C_DIS
LIN {X -0.143,Y -398.764,Z 577.721,A 0.000,B 0.000,C 90.000,E1 165.880} C_DIS
LIN {X 0.174,Y -399.380,Z 577.708,A 0.000,B 0.000,C 90.000,E1 163.378} C_DIS
LIN {X -0.132,Y -400.253,Z 577.694,A 0.000,B 0.000,C 90.000,E1 160.967} C_DIS
LIN {X 0.229,Y -401.356,Z 577.681,A 0.000,B 0.000,C 90.000,E1 158.465} C_DIS
LIN {X 0.014,Y -402.524,Z 577.667,A 0.000,B 0.000,C 90.000,E1 156.049} C_DIS
LIN {X 0.186,Y -403.425,Z 577.657,A 0.000,B 0.000,C 90.000,E1 154.280} C_DIS
LIN {X 0.007,Y -404.351,Z 577.648,A 0.000,B 0.000,C 90.000,E1 152.564} C_DIS
LIN {X -0.038,Y -405.088,Z 577.640,A 0.000,B 0.000,C 90.000,E1 151.179} C_DIS
LIN {X -0.157,Y -405.860,Z 577.630,A 0.000,B 0.000,C 90.000,E1 149.459} C_DIS
LIN {X 0.039,Y -406.393,Z 577.623,A 0.000,B 0.000,C 90.000,E1 148.043} C_DIS
LIN {X 0.059,Y -406.961,Z 577.611,A 0.000,B 0.000,C 90.000,E1 145.960} C_DIS
LIN {X -0.040,Y -407.343,Z 577.601,A 0.000,B 0.000,C 90.000,E1 144.242} C_DIS
LIN {X 0.208,Y -407.671,Z 577.592,A 0.000,B 0.000,C 90.000,E1 142.477} C_DIS
LIN {X 0.231,Y -407.871,Z 577.584,A 0.000,B 0.000,C 90.000,E1 141.090} C_DIS
LIN {X -0.070,Y -408.211,Z 577.573,A 0.000,B 0.000,C 90.000,E1 139.057} C_DIS
LIN {X 0.061,Y -408.462,Z 577.563,A 0.000,B 0.000,C 90.000,E1 137.310} C_DIS
LIN {X -0.004,Y -408.673,Z 577.548,A 0.000,B 0.000,C 90.000,E1 134.555} C_DIS
LIN {X -0.178,Y -408.912,Z 577.538,A 0.000,B 0.000,C 90.000,E1 132.852} C_DIS
LIN {X 0.086,Y -409.055,Z 577.530,A 0.000,B 0.000,C 90.000,E1 131.434} C_DIS
LIN {X -0.192,Y -409.065,Z 577.523,A 0.000,B 0.000,C 90.000,E1 130.092} C_DIS
LIN {X 0.107,Y -408.843,Z 577.515,A 0.000,B 0.000,C 90.000,E1 128.669} C_DIS
LIN {X 0.119,Y -408.808,Z 577.513,A 0.000,B 0.000,C 90.000,E1 128.257} C_DIS
LIN {X -0.013,Y -415.649,Z 577.500,A 0.000,B 0.000,C 90.000,E1 125.931} C_DIS
LIN {X -0.153,Y -425.082,Z 577.479,A 0.000,B 0.000,C 90.000,E1 122.212} C_DIS
LIN {X -0.003,Y -430.069,Z 577.470,A 0.000,B 0.000,C 90.000,E1 120.512} C_DIS
LIN {X -0.223,Y -431.025,Z 577.468,A 0.000,B 0.000,C 90.000,E1 120.207} C_DIS
LIN {X -0.011,Y -433.055,Z 577.463,A 0.000,B 0.000,C 90.000,E1 119.283} C_DIS
LIN {X -0.050,Y -433.076,Z 577.463,A 0.000,B 0.000,C 90.000,E1 119.283} C_DIS
LIN {X -0.047,Y -448.984,Z 577.459,A 0.000,B 0.000,C 90.000,E1 118.565} C_DIS
LIN {X 0.026,Y -469.523,Z 577.453,A 0.000,B 0.000,C 90.000,E1 117.590} C_DIS
LIN {X -0.257,Y -479.650,Z 577.451,A 0.000,B 0.000,C 90.000,E1 117.129} C_DIS
LIN {X -0.258,Y -489.676,Z 577.448,A 0.000,B 0.000,C 90.000,E1 116.616} C_DIS
LIN {X 0.094,Y -499.550,Z 577.445,A 0.000,B 0.000,C 90.000,E1 116.027} C_DIS
LIN {X 0.092,Y -509.264,Z 577.442,A 0.000,B 0.000,C 90.000,E1 115.463} C_DIS
LIN {X -0.160,Y -518.893,Z 577.438,A 0.000,B 0.000,C 90.000,E1 114.899} C_DIS
LIN {X -0.003,Y -530.923,Z 577.434,A 0.000,B 0.000,C 90.000,E1 114.079} C_DIS
LIN {X -0.032,Y -541.134,Z 577.430,A 0.000,B 0.000,C 90.000,E1 113.334} C_DIS
LIN {X -0.223,Y -546.822,Z 577.427,A 0.000,B 0.000,C 90.000,E1 112.898} C_DIS
LIN {X 0.001,Y -551.201,Z 577.425,A 0.000,B 0.000,C 90.000,E1 112.514} C_DIS
LIN {X -0.217,Y -556.214,Z 577.423,A 0.000,B 0.000,C 90.000,E1 112.078} C_DIS
LIN {X -0.095,Y -562.014,Z 577.419,A 0.000,B 0.000,C 90.000,E1 111.461} C_DIS
LIN {X -0.109,Y -566.667,Z 577.416,A 0.000,B 0.000,C 90.000,E1 110.918} C_DIS
LIN {X -0.262,Y -571.776,Z 577.412,A 0.000,B 0.000,C 90.000,E1 110.248} C_DIS
LIN {X 0.084,Y -576.907,Z 577.408,A 0.000,B 0.000,C 90.000,E1 109.396} C_DIS
LIN {X 0.103,Y -580.201,Z 577.405,A 0.000,B 0.000,C 90.000,E1 108.852} C_DIS
LIN {X -0.272,Y -585.110,Z 577.400,A 0.000,B 0.000,C 90.000,E1 107.946} C_DIS
LIN {X 0.214,Y -588.987,Z 577.395,A 0.000,B 0.000,C 90.000,E1 107.094} C_DIS
LIN {X 0.100,Y -592.052,Z 577.391,A 0.000,B 0.000,C 90.000,E1 106.441} C_DIS
LIN {X 0.185,Y -596.556,Z 577.386,A 0.000,B 0.000,C 90.000,E1 105.371} C_DIS
LIN {X 0.329,Y -598.727,Z 577.383,A 0.000,B 0.000,C 90.000,E1 104.828} C_DIS
LIN {X 0.078,Y -603.603,Z 577.375,A 0.000,B 0.000,C 90.000,E1 103.536} C_DIS
LIN {X 0.249,Y -609.348,Z 577.367,A 0.000,B 0.000,C 90.000,E1 101.951} C_DIS
LIN {X -0.072,Y -615.077,Z 577.358,A 0.000,B 0.000,C 90.000,E1 100.423} C_DIS
LIN {X 0.062,Y -618.777,Z 577.352,A 0.000,B 0.000,C 90.000,E1 99.378} C_DIS
LIN {X 0.157,Y -622.360,Z 577.346,A 0.000,B 0.000,C 90.000,E1 98.341} C_DIS
LIN {X -0.226,Y -625.827,Z 577.341,A 0.000,B 0.000,C 90.000,E1 97.352} C_DIS
LIN {X -0.028,Y -629.084,Z 577.335,A 0.000,B 0.000,C 90.000,E1 96.315} C_DIS
LIN {X -0.194,Y -631.397,Z 577.331,A 0.000,B 0.000,C 90.000,E1 95.568} C_DIS
LIN {X -0.279,Y -633.517,Z 577.327,A 0.000,B 0.000,C 90.000,E1 94.816} C_DIS
LIN {X 0.229,Y -635.367,Z 577.322,A 0.000,B 0.000,C 90.000,E1 94.012} C_DIS
LIN {X 0.086,Y -636.961,Z 577.318,A 0.000,B 0.000,C 90.000,E1 93.269} C_DIS
LIN {X -0.249,Y -638.894,Z 577.313,A 0.000,B 0.000,C 90.000,E1 92.293} C_DIS
LIN {X 0.315,Y -640.097,Z 577.308,A 0.000,B 0.000,C 90.000,E1 91.489} C_DIS
LIN {X 0.233,Y -641.072,Z 577.304,A 0.000,B 0.000,C 90.000,E1 90.745} C_DIS
LIN {X 0.162,Y -641.801,Z 577.300,A 0.000,B 0.000,C 90.000,E1 90.000} C_DIS
LIN {X 0.099,Y -642.282,Z 577.296,A 0.000,B 0.000,C 90.000,E1 89.255} C_DIS
LIN {X 0.272,Y -642.432,Z 577.293,A 0.000,B 0.000,C 90.000,E1 88.740} C_DIS
LIN {X 0.232,Y -642.478,Z 577.289,A 0.000,B 0.000,C 90.000,E1 87.993} C_DIS
LIN {X -0.067,Y -642.107,Z 577.283,A 0.000,B 0.000,C 90.000,E1 87.020} C_DIS
LIN {X -0.105,Y -641.638,Z 577.279,A 0.000,B 0.000,C 90.000,E1 86.274} C_DIS
LIN {X 0.247,Y -640.632,Z 577.274,A 0.000,B 0.000,C 90.000,E1 85.241} C_DIS
LIN {X -0.253,Y -639.079,Z 577.267,A 0.000,B 0.000,C 90.000,E1 84.033} C_DIS
LIN {X 0.116,Y -637.431,Z 577.261,A 0.000,B 0.000,C 90.000,E1 82.996} C_DIS
LIN {X -0.257,Y -636.455,Z 577.258,A 0.000,B 0.000,C 90.000,E1 82.527} C_DIS
LIN {X -0.110,Y -633.634,Z 577.251,A 0.000,B 0.000,C 90.000,E1 81.254} C_DIS
LIN {X 0.172,Y -631.095,Z 577.246,A 0.000,B 0.000,C 90.000,E1 80.218} C_DIS
LIN {X 0.012,Y -628.320,Z 577.240,A 0.000,B 0.000,C 90.000,E1 79.218} C_DIS
LIN {X 0.109,Y -624.553,Z 577.233,A 0.000,B 0.000,C 90.000,E1 77.937} C_DIS
LIN {X 0.089,Y -622.081,Z 577.229,A 0.000,B 0.000,C 90.000,E1 77.173} C_DIS
LIN {X 0.265,Y -620.323,Z 577.226,A 0.000,B 0.000,C 90.000,E1 76.645} C_DIS
LIN {X 0.202,Y -617.456,Z 577.222,A 0.000,B 0.000,C 90.000,E1 75.880} C_DIS
LIN {X 0.264,Y -614.495,Z 577.217,A 0.000,B 0.000,C 90.000,E1 75.102} C_DIS
LIN {X 0.139,Y -611.274,Z 577.213,A 0.000,B 0.000,C 90.000,E1 74.338} C_DIS
LIN {X -0.044,Y -606.517,Z 577.207,A 0.000,B 0.000,C 90.000,E1 73.323} C_DIS
LIN {X -0.089,Y -602.570,Z 577.203,A 0.000,B 0.000,C 90.000,E1 72.543} C_DIS
LIN {X -0.166,Y -597.558,Z 577.198,A 0.000,B 0.000,C 90.000,E1 71.638} C_DIS
LIN {X 0.027,Y -593.095,Z 577.194,A 0.000,B 0.000,C 90.000,E1 70.859} C_DIS
LIN {X 0.032,Y -587.802,Z 577.189,A 0.000,B 0.000,C 90.000,E1 70.061} C_DIS
LIN {X 0.122,Y -584.046,Z 577.186,A 0.000,B 0.000,C 90.000,E1 69.518} C_DIS
LIN {X -0.361,Y -579.965,Z 577.183,A 0.000,B 0.000,C 90.000,E1 69.028} C_DIS
LIN {X -0.196,Y -574.189,Z 577.180,A 0.000,B 0.000,C 90.000,E1 68.337} C_DIS
LIN {X 0.213,Y -569.615,Z 577.177,A 0.000,B 0.000,C 90.000,E1 67.794} C_DIS
LIN {X 0.141,Y -564.759,Z 577.174,A 0.000,B 0.000,C 90.000,E1 67.305} C_DIS
LIN {X 0.306,Y -559.439,Z 577.171,A 0.000,B 0.000,C 90.000,E1 66.794} C_DIS
LIN {X 0.081,Y -553.983,Z 577.169,A 0.000,B 0.000,C 90.000,E1 66.357} C_DIS
LIN {X 0.141,Y -549.385,Z 577.167,A 0.000,B 0.000,C 90.000,E1 65.997} C_DIS
LIN {X -0.286,Y -543.035,Z 577.164,A 0.000,B 0.000,C 90.000,E1 65.613} C_DIS
LIN {X 0.058,Y -538.150,Z 577.163,A 0.000,B 0.000,C 90.000,E1 65.281} C_DIS
LIN {X -0.086,Y -529.613,Z 577.160,A 0.000,B 0.000,C 90.000,E1 64.845} C_DIS
LIN {X -0.039,Y -526.223,Z 577.159,A 0.000,B 0.000,C 90.000,E1 64.665} C_DIS
LIN {X 0.101,Y -519.283,Z 577.158,A 0.000,B 0.000,C 90.000,E1 64.332} C_DIS
LIN {X -0.219,Y -514.496,Z 577.156,A 0.000,B 0.000,C 90.000,E1 64.152} C_DIS
LIN {X 0.283,Y -496.873,Z 577.152,A 0.000,B 0.000,C 90.000,E1 63.384} C_DIS
LIN {X -0.052,Y -469.353,Z 577.146,A 0.000,B 0.000,C 90.000,E1 62.281} C_DIS
LIN {X 0.019,Y -462.501,Z 577.144,A 0.000,B 0.000,C 90.000,E1 61.975} C_DIS
LIN {X 0.134,Y -454.807,Z 577.142,A 0.000,B 0.000,C 90.000,E1 61.591} C_DIS
LIN {X 0.093,Y -454.750,Z 577.142,A 0.000,B 0.000,C 90.000,E1 61.591} C_DIS
LIN {X -0.249,Y -445.995,Z 577.120,A 0.000,B 0.000,C 90.000,E1 57.661} C_DIS
LIN {X 0.186,Y -444.225,Z 577.115,A 0.000,B 0.000,C 90.000,E1 56.628} C_DIS
LIN {X -0.125,Y -443.529,Z 577.113,A 0.000,B 0.000,C 90.000,E1 56.342} C_DIS
LIN {X 0.120,Y -436.032,Z 577.095,A 0.000,B 0.000,C 90.000,E1 53.130} C_DIS
LIN {X -0.220,Y -438.244,Z 577.084,A 0.000,B 0.000,C 90.000,E1 51.090} C_DIS
LIN {X 0.262,Y -439.992,Z 577.075,A 0.000,B 0.000,C 90.000,E1 49.380} C_DIS
LIN {X -0.216,Y -442.085,Z 577.064,A 0.000,B 0.000,C 90.000,E1 47.472} C_DIS
LIN {X -0.026,Y -443.810,Z 577.055,A 0.000,B 0.000,C 90.000,E1 45.810} C_DIS
LIN {X -0.103,Y -445.003,Z 577.047,A 0.000,B 0.000,C 90.000,E1 44.514} C_DIS
LIN {X -0.150,Y -445.805,Z 577.042,A 0.000,B 0.000,C 90.000,E1 43.542} C_DIS
LIN {X 0.133,Y -446.484,Z 577.036,A 0.000,B 0.000,C 90.000,E1 42.528} C_DIS
LIN {X 0.103,Y -447.321,Z 577.027,A 0.000,B 0.000,C 90.000,E1 40.906} C_DIS
LIN {X 0.108,Y -447.738,Z 577.022,A 0.000,B 0.000,C 90.000,E1 39.930} C_DIS
LIN {X 0.166,Y -448.130,Z 577.015,A 0.000,B 0.000,C 90.000,E1 38.624} C_DIS
LIN {X -0.119,Y -448.363,Z 577.008,A 0.000,B 0.000,C 90.000,E1 37.363} C_DIS
LIN {X 0.306,Y -448.454,Z 577.000,A 0.000,B 0.000,C 90.000,E1 36.011} C_DIS
LIN {X -0.124,Y -448.203,Z 576.990,A 0.000,B 0.000,C 90.000,E1 34.119} C_DIS
LIN {X 0.254,Y -447.849,Z 576.977,A 0.000,B 0.000,C 90.000,E1 31.799} C_DIS
LIN {X 0.008,Y -447.695,Z 576.968,A 0.000,B 0.000,C 90.000,E1 30.207} C_DIS
LIN {X 0.151,Y -447.547,Z 576.959,A 0.000,B 0.000,C 90.000,E1 28.565} C_DIS
LIN {X 0.081,Y -447.379,Z 576.950,A 0.000,B 0.000,C 90.000,E1 26.950} C_DIS
LIN {X -0.132,Y -447.192,Z 576.939,A 0.000,B 0.000,C 90.000,E1 25.027} C_DIS
LIN {X -0.009,Y -447.203,Z 576.930,A 0.000,B 0.000,C 90.000,E1 23.387} C_DIS
LIN {X 0.088,Y -447.316,Z 576.917,A 0.000,B 0.000,C 90.000,E1 21.099} C_DIS
LIN {X 0.153,Y -447.464,Z 576.906,A 0.000,B 0.000,C 90.000,E1 19.141} C_DIS
LIN {X 0.088,Y -447.802,Z 576.892,A 0.000,B 0.000,C 90.000,E1 16.551} C_DIS
LIN {X 0.178,Y -448.348,Z 576.881,A 0.000,B 0.000,C 90.000,E1 14.592} C_DIS
LIN {X 0.108,Y -449.321,Z 576.867,A 0.000,B 0.000,C 90.000,E1 12.007} C_DIS
LIN {X 0.220,Y -450.460,Z 576.854,A 0.000,B 0.000,C 90.000,E1 9.726} C_DIS
LIN {X -0.196,Y -451.476,Z 576.845,A 0.000,B 0.000,C 90.000,E1 8.163} C_DIS
LIN {X -0.090,Y -453.285,Z 576.831,A 0.000,B 0.000,C 90.000,E1 5.568} C_DIS
LIN {X -0.170,Y -455.241,Z 576.818,A 0.000,B 0.000,C 90.000,E1 3.326} C_DIS
LIN {X 0.041,Y -457.089,Z 576.808,A 0.000,B 0.000,C 90.000,E1 1.375} C_DIS
LIN {X -0.090,Y -459.261,Z 576.797,A 0.000,B 0.000,C 90.000,E1 359.484} C_DIS
LIN {X 0.148,Y -462.524,Z 576.783,A 0.000,B 0.000,C 90.000,E1 356.906} C_DIS
LIN {X 0.108,Y -465.241,Z 576.772,A 0.000,B 0.000,C 90.000,E1 355.008} C_DIS
LIN {X -0.060,Y -468.536,Z 576.760,A 0.000,B 0.000,C 90.000,E1 352.818} C_DIS
LIN {X 0.055,Y -470.446,Z 576.753,A 0.000,B 0.000,C 90.000,E1 351.546} C_DIS
LIN {X 0.023,Y -472.857,Z 576.744,A 0.000,B 0.000,C 90.000,E1 349.982} C_DIS
LIN {X -0.053,Y -475.721,Z 576.734,A 0.000,B 0.000,C 90.000,E1 348.117} C_DIS
LIN {X -0.011,Y -479.209,Z 576.722,A 0.000,B 0.000,C 90.000,E1 345.936} C_DIS
LIN {X -0.050,Y -481.923,Z 576.713,A 0.000,B 0.000,C 90.000,E1 344.393} C_DIS
LIN {X -0.043,Y -485.330,Z 576.703,A 0.000,B 0.000,C 90.000,E1 342.543} C_DIS
LIN {X 0.203,Y -489.493,Z 576.691,A 0.000,B 0.000,C 90.000,E1 340.369} C_DIS
LIN {X -0.239,Y -492.999,Z 576.681,A 0.000,B 0.000,C 90.000,E1 338.592} C_DIS
LIN {X -0.065,Y -495.269,Z 576.674,A 0.000,B 0.000,C 90.000,E1 337.358} C_DIS
LIN {X -0.318,Y -497.460,Z 576.667,A 0.000,B 0.000,C 90.000,E1 336.177} C_DIS
LIN {X -0.274,Y -500.000,Z 576.659,A 0.000,B 0.000,C 90.000,E1 334.665} C_DIS
LIN {X -0.031,Y -502.026,Z 576.652,A 0.000,B 0.000,C 90.000,E1 333.435} C_DIS
LIN {X -0.123,Y -504.380,Z 576.644,A 0.000,B 0.000,C 90.000,E1 331.948} C_DIS
LIN {X -0.178,Y -506.724,Z 576.636,A 0.000,B 0.000,C 90.000,E1 330.461} C_DIS
LIN {X -0.056,Y -509.676,Z 576.626,A 0.000,B 0.000,C 90.000,E1 328.663} C_DIS
LIN {X -0.308,Y -512.636,Z 576.616,A 0.000,B 0.000,C 90.000,E1 326.914} C_DIS
LIN {X -0.003,Y -516.221,Z 576.605,A 0.000,B 0.000,C 90.000,E1 324.815} C_DIS
LIN {X 0.098,Y -518.854,Z 576.596,A 0.000,B 0.000,C 90.000,E1 323.336} C_DIS
LIN {X -0.040,Y -523.733,Z 576.582,A 0.000,B 0.000,C 90.000,E1 320.723} C_DIS
LIN {X 0.086,Y -531.846,Z 576.561,A 0.000,B 0.000,C 90.000,E1 316.944} C_DIS
LIN {X -0.061,Y -534.888,Z 576.555,A 0.000,B 0.000,C 90.000,E1 315.810} C_DIS
LIN {X 0.062,Y -537.367,Z 576.551,A 0.000,B 0.000,C 90.000,E1 315.081} C_DIS
LIN {X -0.024,Y -539.395,Z 576.548,A 0.000,B 0.000,C 90.000,E1 314.636} C_DIS
LIN {X -0.220,Y -540.230,Z 576.547,A 0.000,B 0.000,C 90.000,E1 314.514} C_DIS
LIN {X -0.221,Y -541.381,Z 576.546,A 0.000,B 0.000,C 90.000,E1 314.352} C_DIS
LIN {X 0.155,Y -543.197,Z 576.545,A 0.000,B 0.000,C 90.000,E1 314.028} C_DIS
LIN {X 0.156,Y -544.650,Z 576.544,A 0.000,B 0.000,C 90.000,E1 313.866} C_DIS
LIN {X -0.219,Y -546.929,Z 576.542,A 0.000,B 0.000,C 90.000,E1 313.623} C_DIS
LIN {X -0.100,Y -551.209,Z 576.540,A 0.000,B 0.000,C 90.000,E1 313.176} C_DIS
LIN {X 0.121,Y -554.509,Z 576.538,A 0.000,B 0.000,C 90.000,E1 312.852} C_DIS
LIN {X -0.008,Y -562.567,Z 576.535,A 0.000,B 0.000,C 90.000,E1 312.243} C_DIS
LIN {X -0.053,Y -578.778,Z 576.528,A 0.000,B 0.000,C 90.000,E1 311.067} C_DIS
LIN {X 0.287,Y -591.967,Z 576.523,A 0.000,B 0.000,C 90.000,E1 310.092} C_DIS
LIN {X 0.014,Y -597.637,Z 576.521,A 0.000,B 0.000,C 90.000,E1 309.688} C_DIS
LIN {X -0.017,Y -603.169,Z 576.518,A 0.000,B 0.000,C 90.000,E1 309.241} C_DIS
LIN {X 0.191,Y -608.426,Z 576.515,A 0.000,B 0.000,C 90.000,E1 308.749} C_DIS
LIN {X -0.234,Y -613.489,Z 576.513,A 0.000,B 0.000,C 90.000,E1 308.302} C_DIS
LIN {X -0.351,Y -618.315,Z 576.510,A 0.000,B 0.000,C 90.000,E1 307.810} C_DIS
LIN {X 0.306,Y -622.974,Z 576.507,A 0.000,B 0.000,C 90.000,E1 307.237} C_DIS
LIN {X -0.055,Y -629.572,Z 576.503,A 0.000,B 0.000,C 90.000,E1 306.503} C_DIS
LIN {X -0.221,Y -633.740,Z 576.500,A 0.000,B 0.000,C 90.000,E1 306.011} C_DIS
LIN {X 0.054,Y -641.410,Z 576.494,A 0.000,B 0.000,C 90.000,E1 304.978} C_DIS
LIN {X -0.031,Y -645.027,Z 576.492,A 0.000,B 0.000,C 90.000,E1 304.485} C_DIS
LIN {X -0.062,Y -649.150,Z 576.488,A 0.000,B 0.000,C 90.000,E1 303.865} C_DIS
LIN {X -0.137,Y -651.500,Z 576.486,A 0.000,B 0.000,C 90.000,E1 303.499} C_DIS
LIN {X 0.341,Y -653.557,Z 576.484,A 0.000,B 0.000,C 90.000,E1 303.086} C_DIS
LIN {X -0.073,Y -655.613,Z 576.482,A 0.000,B 0.000,C 90.000,E1 302.752} C_DIS
LIN {X -0.024,Y -658.658,Z 576.479,A 0.000,B 0.000,C 90.000,E1 302.133} C_DIS
LIN {X -0.359,Y -660.949,Z 576.476,A 0.000,B 0.000,C 90.000,E1 301.671} C_DIS
LIN {X -0.211,Y -664.187,Z 576.472,A 0.000,B 0.000,C 90.000,E1 300.924} C_DIS
LIN {X -0.077,Y -665.137,Z 576.470,A 0.000,B 0.000,C 90.000,E1 300.669} C_DIS
LIN {X 0.064,Y -666.306,Z 576.469,A 0.000,B 0.000,C 90.000,E1 300.413} C_DIS
LIN {X 0.264,Y -669.326,Z 576.465,A 0.000,B 0.000,C 90.000,E1 299.667} C_DIS
LIN {X -0.262,Y -672.983,Z 576.460,A 0.000,B 0.000,C 90.000,E1 298.743} C_DIS
LIN {X 0.263,Y -675.460,Z 576.456,A 0.000,B 0.000,C 90.000,E1 297.975} C_DIS
LIN {X -0.153,Y -676.187,Z 576.454,A 0.000,B 0.000,C 90.000,E1 297.769} C_DIS
LIN {X 0.031,Y -677.097,Z 576.453,A 0.000,B 0.000,C 90.000,E1 297.513} C_DIS
LIN {X -0.196,Y -678.589,Z 576.450,A 0.000,B 0.000,C 90.000,E1 297.052} C_DIS
LIN {X -0.003,Y -679.492,Z 576.449,A 0.000,B 0.000,C 90.000,E1 296.796} C_DIS
LIN {X 0.192,Y -680.069,Z 576.448,A 0.000,B 0.000,C 90.000,E1 296.539} C_DIS
LIN {X -0.321,Y -680.870,Z 576.445,A 0.000,B 0.000,C 90.000,E1 296.104} C_DIS
LIN {X -0.118,Y -681.000,Z 576.444,A 0.000,B 0.000,C 90.000,E1 295.848} C_DIS
LIN {X 0.085,Y -680.905,Z 576.442,A 0.000,B 0.000,C 90.000,E1 295.591} C_DIS
LIN {X 0.287,Y -680.604,Z 576.441,A 0.000,B 0.000,C 90.000,E1 295.335} C_DIS
LIN {X -0.415,Y -679.838,Z 576.440,A 0.000,B 0.000,C 90.000,E1 295.155} C_DIS
LIN {X -0.017,Y -676.534,Z 576.437,A 0.000,B 0.000,C 90.000,E1 294.643} C_DIS
LIN {X -0.366,Y -674.543,Z 576.436,A 0.000,B 0.000,C 90.000,E1 294.463} C_DIS
LIN {X -0.120,Y -667.354,Z 576.433,A 0.000,B 0.000,C 90.000,E1 294.027} C_DIS
LIN {X -0.271,Y -665.235,Z 576.433,A 0.000,B 0.000,C 90.000,E1 293.951} C_DIS
LIN {X 0.184,Y -662.690,Z 576.432,A 0.000,B 0.000,C 90.000,E1 293.823} C_DIS
LIN {X 0.046,Y -653.087,Z 576.431,A 0.000,B 0.000,C 90.000,E1 293.567} C_DIS
LIN {X -0.088,Y -630.433,Z 576.428,A 0.000,B 0.000,C 90.000,E1 293.078} C_DIS
LIN {X 0.135,Y -616.792,Z 576.426,A 0.000,B 0.000,C 90.000,E1 292.717} C_DIS
LIN {X -0.242,Y -596.795,Z 576.423,A 0.000,B 0.000,C 90.000,E1 292.153} C_DIS
LIN {X -0.164,Y -572.794,Z 576.419,A 0.000,B 0.000,C 90.000,E1 291.354} C_DIS
LIN {X -0.270,Y -566.609,Z 576.417,A 0.000,B 0.000,C 90.000,E1 291.099} C_DIS
LIN {X -0.146,Y -563.462,Z 576.416,A 0.000,B 0.000,C 90.000,E1 290.844} C_DIS
LIN {X -0.181,Y -563.420,Z 576.416,A 0.000,B 0.000,C 90.000,E1 290.844} C_DIS
LIN {X 0.045,Y -562.707,Z 576.415,A 0.000,B 0.000,C 90.000,E1 290.663} C_DIS
LIN {X -0.208,Y -562.445,Z 576.414,A 0.000,B 0.000,C 90.000,E1 290.482} C_DIS
LIN {X 0.110,Y -562.259,Z 576.412,A 0.000,B 0.000,C 90.000,E1 290.174} C_DIS
LIN {X 0.249,Y -562.368,Z 576.405,A 0.000,B 0.000,C 90.000,E1 288.779} C_DIS
LIN {X 0.217,Y -562.032,Z 576.397,A 0.000,B 0.000,C 90.000,E1 287.402} C_DIS
LIN {X 0.181,Y -561.508,Z 576.389,A 0.000,B 0.000,C 90.000,E1 286.024} C_DIS
LIN {X -0.015,Y -560.788,Z 576.381,A 0.000,B 0.000,C 90.000,E1 284.662} C_DIS
LIN {X -0.223,Y -559.975,Z 576.374,A 0.000,B 0.000,C 90.000,E1 283.300} C_DIS
LIN {X 0.231,Y -559.034,Z 576.365,A 0.000,B 0.000,C 90.000,E1 281.591} C_DIS
LIN {X -0.253,Y -558.227,Z 576.357,A 0.000,B 0.000,C 90.000,E1 280.254} C_DIS
LIN {X 0.129,Y -557.018,Z 576.345,A 0.000,B 0.000,C 90.000,E1 277.992} C_DIS
LIN {X 0.088,Y -556.471,Z 576.337,A 0.000,B 0.000,C 90.000,E1 276.606} C_DIS
LIN {X -0.271,Y -555.635,Z 576.324,A 0.000,B 0.000,C 90.000,E1 274.416} C_DIS
LIN {X -0.185,Y -554.922,Z 576.312,A 0.000,B 0.000,C 90.000,E1 272.178} C_DIS
LIN {X 0.268,Y -554.354,Z 576.303,A 0.000,B 0.000,C 90.000,E1 270.458} C_DIS
LIN {X 0.141,Y -553.637,Z 576.293,A 0.000,B 0.000,C 90.000,E1 268.797} C_DIS
LIN {X 0.099,Y -552.823,Z 576.283,A 0.000,B 0.000,C 90.000,E1 266.846} C_DIS
LIN {X -0.114,Y -552.180,Z 576.275,A 0.000,B 0.000,C 90.000,E1 265.469} C_DIS
LIN {X 0.244,Y -551.404,Z 576.267,A 0.000,B 0.000,C 90.000,E1 264.033} C_DIS
LIN {X 0.094,Y -550.485,Z 576.259,A 0.000,B 0.000,C 90.000,E1 262.648} C_DIS
LIN {X -0.205,Y -549.725,Z 576.255,A 0.000,B 0.000,C 90.000,E1 261.837} C_DIS
LIN {X 0.239,Y -548.294,Z 576.247,A 0.000,B 0.000,C 90.000,E1 260.387} C_DIS
LIN {X 0.210,Y -546.624,Z 576.237,A 0.000,B 0.000,C 90.000,E1 258.701} C_DIS
LIN {X 0.152,Y -545.210,Z 576.230,A 0.000,B 0.000,C 90.000,E1 257.297} C_DIS
LIN {X -0.251,Y -543.411,Z 576.220,A 0.000,B 0.000,C 90.000,E1 255.644} C_DIS
LIN {X -0.319,Y -542.236,Z 576.214,A 0.000,B 0.000,C 90.000,E1 254.519} C_DIS
LIN {X 0.196,Y -541.278,Z 576.209,A 0.000,B 0.000,C 90.000,E1 253.614} C_DIS
LIN {X -0.203,Y -539.500,Z 576.201,A 0.000,B 0.000,C 90.000,E1 252.236} C_DIS
LIN {X -0.174,Y -537.924,Z 576.195,A 0.000,B 0.000,C 90.000,E1 251.094} C_DIS
LIN {X -0.208,Y -536.601,Z 576.190,A 0.000,B 0.000,C 90.000,E1 250.242} C_DIS
LIN {X 0.160,Y -534.171,Z 576.182,A 0.000,B 0.000,C 90.000,E1 248.773} C_DIS
LIN {X 0.077,Y -532.543,Z 576.177,A 0.000,B 0.000,C 90.000,E1 247.922} C_DIS
LIN {X -0.121,Y -530.189,Z 576.171,A 0.000,B 0.000,C 90.000,E1 246.794} C_DIS
LIN {X -0.169,Y -527.166,Z 576.163,A 0.000,B 0.000,C 90.000,E1 245.357} C_DIS
LIN {X 0.257,Y -524.626,Z 576.157,A 0.000,B 0.000,C 90.000,E1 244.152} C_DIS
LIN {X 0.172,Y -521.975,Z 576.150,A 0.000,B 0.000,C 90.000,E1 242.999} C_DIS
LIN {X -0.087,Y -519.902,Z 576.145,A 0.000,B 0.000,C 90.000,E1 242.153} C_DIS
LIN {X 0.090,Y -517.733,Z 576.140,A 0.000,B 0.000,C 90.000,E1 241.257} C_DIS
LIN {X 0.038,Y -515.464,Z 576.136,A 0.000,B 0.000,C 90.000,E1 240.383} C_DIS
LIN {X 0.061,Y -512.212,Z 576.129,A 0.000,B 0.000,C 90.000,E1 239.203} C_DIS
LIN {X -0.175,Y -507.323,Z 576.119,A 0.000,B 0.000,C 90.000,E1 237.454} C_DIS
LIN {X -0.135,Y -503.176,Z 576.111,A 0.000,B 0.000,C 90.000,E1 235.960} C_DIS
LIN {X -0.306,Y -498.919,Z 576.103,A 0.000,B 0.000,C 90.000,E1 234.482} C_DIS
LIN {X -0.130,Y -491.542,Z 576.087,A 0.000,B 0.000,C 90.000,E1 231.743} C_DIS
LIN {X -0.105,Y -485.159,Z 576.074,A 0.000,B 0.000,C 90.000,E1 229.299} C_DIS
LIN {X -0.132,Y -479.681,Z 576.062,A 0.000,B 0.000,C 90.000,E1 227.148} C_DIS
LIN {X 0.240,Y -475.123,Z 576.052,A 0.000,B 0.000,C 90.000,E1 225.243} C_DIS
LIN {X 0.161,Y -470.654,Z 576.041,A 0.000,B 0.000,C 90.000,E1 223.380} C_DIS
LIN {X -0.005,Y -466.345,Z 576.031,A 0.000,B 0.000,C 90.000,E1 221.515} C_DIS
LIN {X 0.180,Y -461.523,Z 576.018,A 0.000,B 0.000,C 90.000,E1 219.277} C_DIS
LIN {X 0.209,Y -457.431,Z 576.008,A 0.000,B 0.000,C 90.000,E1 217.363} C_DIS
LIN {X -0.133,Y -454.119,Z 575.999,A 0.000,B 0.000,C 90.000,E1 215.804} C_DIS
LIN {X -0.042,Y -448.927,Z 575.985,A 0.000,B 0.000,C 90.000,E1 213.214} C_DIS
LIN {X 0.144,Y -444.073,Z 575.970,A 0.000,B 0.000,C 90.000,E1 210.590} C_DIS
LIN {X 0.200,Y -441.129,Z 575.961,A 0.000,B 0.000,C 90.000,E1 208.949} C_DIS
LIN {X -0.008,Y -438.282,Z 575.952,A 0.000,B 0.000,C 90.000,E1 207.334} C_DIS
LIN {X 0.137,Y -434.849,Z 575.941,A 0.000,B 0.000,C 90.000,E1 205.335} C_DIS
LIN {X 0.004,Y -432.057,Z 575.932,A 0.000,B 0.000,C 90.000,E1 203.695} C_DIS
LIN {X 0.042,Y -429.378,Z 575.922,A 0.000,B 0.000,C 90.000,E1 202.025} C_DIS
LIN {X 0.022,Y -425.910,Z 575.909,A 0.000,B 0.000,C 90.000,E1 199.685} C_DIS
LIN {X -0.169,Y -423.067,Z 575.898,A 0.000,B 0.000,C 90.000,E1 197.692} C_DIS
LIN {X 0.080,Y -419.561,Z 575.883,A 0.000,B 0.000,C 90.000,E1 194.954} C_DIS
LIN {X 0.107,Y -417.843,Z 575.876,A 0.000,B 0.000,C 90.000,E1 193.592} C_DIS
LIN {X 0.011,Y -415.877,Z 575.868,A 0.000,B 0.000,C 90.000,E1 192.243} C_DIS
LIN {X 0.092,Y -411.710,Z 575.851,A 0.000,B 0.000,C 90.000,E1 189.151} C_DIS
LIN {X -0.181,Y -409.331,Z 575.839,A 0.000,B 0.000,C 90.000,E1 187.125} C_DIS
LIN {X -0.156,Y -406.985,Z 575.828,A 0.000,B 0.000,C 90.000,E1 185.049} C_DIS
LIN {X 0.031,Y -403.164,Z 575.807,A 0.000,B 0.000,C 90.000,E1 181.203} C_DIS
LIN {X 0.179,Y -401.411,Z 575.793,A 0.000,B 0.000,C 90.000,E1 178.740} C_DIS
LIN {X -0.052,Y -400.182,Z 575.782,A 0.000,B 0.000,C 90.000,E1 176.674} C_DIS
LIN {X -0.041,Y -398.960,Z 575.762,A 0.000,B 0.000,C 90.000,E1 173.166} C_DIS
LIN {X 0.126,Y -398.555,Z 575.745,A 0.000,B 0.000,C 90.000,E1 169.982} C_DIS
LIN {X 0.162,Y -398.769,Z 575.725,A 0.000,B 0.000,C 90.000,E1 166.464} C_DIS
LIN {X -0.039,Y -399.446,Z 575.709,A 0.000,B 0.000,C 90.000,E1 163.685} C_DIS
LIN {X 0.028,Y -400.265,Z 575.696,A 0.000,B 0.000,C 90.000,E1 161.221} C_DIS
LIN {X -0.079,Y -401.204,Z 575.684,A 0.000,B 0.000,C 90.000,E1 159.135} C_DIS
LIN {X -0.161,Y -402.201,Z 575.672,A 0.000,B 0.000,C 90.000,E1 157.050} C_DIS
LIN {X 0.084,Y -403.298,Z 575.661,A 0.000,B 0.000,C 90.000,E1 154.921} C_DIS
LIN {X -0.097,Y -404.196,Z 575.651,A 0.000,B 0.000,C 90.000,E1 153.204} C_DIS
LIN {X 0.113,Y -405.154,Z 575.641,A 0.000,B 0.000,C 90.000,E1 151.435} C_DIS
LIN {X -0.206,Y -405.971,Z 575.632,A 0.000,B 0.000,C 90.000,E1 149.744} C_DIS
LIN {X -0.014,Y -406.501,Z 575.624,A 0.000,B 0.000,C 90.000,E1 148.329} C_DIS
LIN {X 0.097,Y -407.018,Z 575.614,A 0.000,B 0.000,C 90.000,E1 146.580} C_DIS
LIN {X 0.095,Y -407.452,Z 575.605,A 0.000,B 0.000,C 90.000,E1 144.848} C_DIS
LIN {X 0.009,Y -407.791,Z 575.595,A 0.000,B 0.000,C 90.000,E1 143.130} C_DIS
LIN {X -0.071,Y -408.058,Z 575.586,A 0.000,B 0.000,C 90.000,E1 141.412} C_DIS
LIN {X 0.200,Y -408.361,Z 575.574,A 0.000,B 0.000,C 90.000,E1 139.299} C_DIS
LIN {X -0.237,Y -408.506,Z 575.568,A 0.000,B 0.000,C 90.000,E1 138.324} C_DIS
LIN {X 0.166,Y -408.638,Z 575.559,A 0.000,B 0.000,C 90.000,E1 136.539} C_DIS
LIN {X 0.257,Y -408.889,Z 575.545,A 0.000,B 0.000,C 90.000,E1 134.109} C_DIS
LIN {X -0.207,Y -409.148,Z 575.536,A 0.000,B 0.000,C 90.000,E1 132.447} C_DIS
LIN {X -0.061,Y -409.196,Z 575.526,A 0.000,B 0.000,C 90.000,E1 130.701} C_DIS
LIN {X 0.090,Y -409.143,Z 575.520,A 0.000,B 0.000,C 90.000,E1 129.644} C_DIS
LIN {X -0.020,Y -408.970,Z 575.515,A 0.000,B 0.000,C 90.000,E1 128.624} C_DIS
LIN {X 0.080,Y -408.919,Z 575.512,A 0.000,B 0.000,C 90.000,E1 128.222} C_DIS
LIN {X -0.125,Y -415.800,Z 575.499,A 0.000,B 0.000,C 90.000,E1 125.884} C_DIS
LIN {X -0.019,Y -425.254,Z 575.479,A 0.000,B 0.000,C 90.000,E1 122.133} C_DIS
LIN {X -0.086,Y -430.258,Z 575.469,A 0.000,B 0.000,C 90.000,E1 120.463} C_DIS
LIN {X -0.087,Y -431.158,Z 575.467,A 0.000,B 0.000,C 90.000,E1 120.129} C_DIS
LIN {X 0.109,Y -433.687,Z 575.461,A 0.000,B 0.000,C 90.000,E1 118.999} C_DIS
LIN {X 0.070,Y -433.763,Z 575.461,A 0.000,B 0.000,C 90.000,E1 118.999} C_DIS
LIN {X 0.035,Y -449.261,Z 575.457,A 0.000,B 0.000,C 90.000,E1 118.309} C_DIS
LIN {X -0.036,Y -468.047,Z 575.452,A 0.000,B 0.000,C 90.000,E1 117.436} C_DIS
LIN {X 0.215,Y -476.500,Z 575.450,A 0.000,B 0.000,C 90.000,E1 117.001} C_DIS
LIN {X -0.107,Y -490.085,Z 575.446,A 0.000,B 0.000,C 90.000,E1 116.360} C_DIS
LIN {X 0.013,Y -501.467,Z 575.443,A 0.000,B 0.000,C 90.000,E1 115.720} C_DIS
LIN {X -0.024,Y -511.176,Z 575.440,A 0.000,B 0.000,C 90.000,E1 115.155} C_DIS
LIN {X -0.124,Y -518.930,Z 575.437,A 0.000,B 0.000,C 90.000,E1 114.695} C_DIS
LIN {X -0.094,Y -528.423,Z 575.434,A 0.000,B 0.000,C 90.000,E1 114.079} C_DIS
LIN {X 0.285,Y -535.791,Z 575.431,A 0.000,B 0.000,C 90.000,E1 113.515} C_DIS
LIN {X 0.133,Y -540.322,Z 575.429,A 0.000,B 0.000,C 90.000,E1 113.206} C_DIS
LIN {X 0.116,Y -545.937,Z 575.427,A 0.000,B 0.000,C 90.000,E1 112.770} C_DIS
LIN {X -0.309,Y -550.393,Z 575.425,A 0.000,B 0.000,C 90.000,E1 112.461} C_DIS
LIN {X -0.124,Y -555.879,Z 575.422,A 0.000,B 0.000,C 90.000,E1 111.950} C_DIS
LIN {X 0.091,Y -561.083,Z 575.419,A 0.000,B 0.000,C 90.000,E1 111.408} C_DIS
LIN {X 0.077,Y -565.915,Z 575.416,A 0.000,B 0.000,C 90.000,E1 110.865} C_DIS
LIN {X 0.119,Y -571.225,Z 575.412,A 0.000,B 0.000,C 90.000,E1 110.174} C_DIS
LIN {X 0.004,Y -575.684,Z 575.408,A 0.000,B 0.000,C 90.000,E1 109.504} C_DIS
LIN {X -0.077,Y -579.875,Z 575.405,A 0.000,B 0.000,C 90.000,E1 108.833} C_DIS
LIN {X -0.226,Y -584.219,Z 575.400,A 0.000,B 0.000,C 90.000,E1 108.055} C_DIS
LIN {X 0.071,Y -588.251,Z 575.396,A 0.000,B 0.000,C 90.000,E1 107.221} C_DIS
LIN {X -0.148,Y -592.039,Z 575.391,A 0.000,B 0.000,C 90.000,E1 106.441} C_DIS
LIN {X 0.239,Y -595.537,Z 575.387,A 0.000,B 0.000,C 90.000,E1 105.607} C_DIS
LIN {X 0.082,Y -598.865,Z 575.382,A 0.000,B 0.000,C 90.000,E1 104.828} C_DIS
LIN {X -0.168,Y -603.866,Z 575.375,A 0.000,B 0.000,C 90.000,E1 103.536} C_DIS
LIN {X -0.328,Y -608.734,Z 575.368,A 0.000,B 0.000,C 90.000,E1 102.243} C_DIS
LIN {X -0.060,Y -614.577,Z 575.359,A 0.000,B 0.000,C 90.000,E1 100.658} C_DIS
LIN {X 0.106,Y -620.150,Z 575.351,A 0.000,B 0.000,C 90.000,E1 99.095} C_DIS
LIN {X -0.221,Y -625.574,Z 575.342,A 0.000,B 0.000,C 90.000,E1 97.587} C_DIS
LIN {X -0.242,Y -629.692,Z 575.335,A 0.000,B 0.000,C 90.000,E1 96.315} C_DIS
LIN {X -0.122,Y -631.299,Z 575.332,A 0.000,B 0.000,C 90.000,E1 95.796} C_DIS
LIN {X 0.148,Y -634.160,Z 575.327,A 0.000,B 0.000,C 90.000,E1 94.759} C_DIS
LIN {X 0.031,Y -636.027,Z 575.322,A 0.000,B 0.000,C 90.000,E1 94.012} C_DIS
LIN {X -0.106,Y -637.645,Z 575.318,A 0.000,B 0.000,C 90.000,E1 93.269} C_DIS
LIN {X 0.207,Y -639.604,Z 575.313,A 0.000,B 0.000,C 90.000,E1 92.236} C_DIS
LIN {X 0.139,Y -640.805,Z 575.308,A 0.000,B 0.000,C 90.000,E1 91.489} C_DIS
LIN {X 0.063,Y -641.791,Z 575.304,A 0.000,B 0.000,C 90.000,E1 90.745} C_DIS
LIN {X 0.000,Y -642.530,Z 575.300,A 0.000,B 0.000,C 90.000,E1 90.000} C_DIS
LIN {X -0.289,Y -643.119,Z 575.294,A 0.000,B 0.000,C 90.000,E1 89.026} C_DIS
LIN {X 0.089,Y -643.165,Z 575.289,A 0.000,B 0.000,C 90.000,E1 87.993} C_DIS
LIN {X -0.202,Y -642.787,Z 575.283,A 0.000,B 0.000,C 90.000,E1 87.020} C_DIS
LIN {X -0.234,Y -642.297,Z 575.279,A 0.000,B 0.000,C 90.000,E1 86.274} C_DIS
LIN {X 0.129,Y -641.253,Z 575.274,A 0.000,B 0.000,C 90.000,E1 85.241} C_DIS
LIN {X -0.108,Y -639.980,Z 575.268,A 0.000,B 0.000,C 90.000,E1 84.261} C_DIS
LIN {X 0.087,Y -639.257,Z 575.265,A 0.000,B 0.000,C 90.000,E1 83.742} C_DIS
LIN {X -0.170,Y -637.508,Z 575.260,A 0.000,B 0.000,C 90.000,E1 82.761} C_DIS
LIN {X -0.177,Y -635.859,Z 575.256,A 0.000,B 0.000,C 90.000,E1 82.008} C_DIS
LIN {X 0.143,Y -633.494,Z 575.250,A 0.000,B 0.000,C 90.000,E1 80.971} C_DIS
LIN {X -0.102,Y -630.826,Z 575.244,A 0.000,B 0.000,C 90.000,E1 79.982} C_DIS
LIN {X 0.035,Y -627.158,Z 575.237,A 0.000,B 0.000,C 90.000,E1 78.701} C_DIS
LIN {X -0.167,Y -623.983,Z 575.232,A 0.000,B 0.000,C 90.000,E1 77.701} C_DIS
LIN {X -0.189,Y -621.390,Z 575.227,A 0.000,B 0.000,C 90.000,E1 76.937} C_DIS
LIN {X -0.238,Y -618.565,Z 575.223,A 0.000,B 0.000,C 90.000,E1 76.172} C_DIS
LIN {X -0.317,Y -615.557,Z 575.219,A 0.000,B 0.000,C 90.000,E1 75.408} C_DIS
LIN {X -0.270,Y -612.320,Z 575.215,A 0.000,B 0.000,C 90.000,E1 74.629} C_DIS
LIN {X -0.209,Y -609.360,Z 575.211,A 0.000,B 0.000,C 90.000,E1 73.976} C_DIS
LIN {X -0.169,Y -605.592,Z 575.207,A 0.000,B 0.000,C 90.000,E1 73.196} C_DIS
LIN {X -0.221,Y -601.510,Z 575.202,A 0.000,B 0.000,C 90.000,E1 72.417} C_DIS
LIN {X -0.264,Y -597.871,Z 575.199,A 0.000,B 0.000,C 90.000,E1 71.764} C_DIS
LIN {X -0.101,Y -594.622,Z 575.196,A 0.000,B 0.000,C 90.000,E1 71.221} C_DIS
LIN {X -0.211,Y -593.048,Z 575.194,A 0.000,B 0.000,C 90.000,E1 70.967} C_DIS
LIN {X -0.027,Y -588.664,Z 575.191,A 0.000,B 0.000,C 90.000,E1 70.296} C_DIS
LIN {X 0.008,Y -584.040,Z 575.187,A 0.000,B 0.000,C 90.000,E1 69.645} C_DIS
LIN {X 0.274,Y -579.859,Z 575.184,A 0.000,B 0.000,C 90.000,E1 69.082} C_DIS
LIN {X 0.220,Y -574.005,Z 575.180,A 0.000,B 0.000,C 90.000,E1 68.411} C_DIS
LIN {X -0.259,Y -568.959,Z 575.177,A 0.000,B 0.000,C 90.000,E1 67.922} C_DIS
LIN {X 0.244,Y -563.754,Z 575.174,A 0.000,B 0.000,C 90.000,E1 67.358} C_DIS
LIN {X -0.344,Y -559.774,Z 575.172,A 0.000,B 0.000,C 90.000,E1 67.050} C_DIS
LIN {X -0.083,Y -553.904,Z 575.170,A 0.000,B 0.000,C 90.000,E1 66.538} C_DIS
LIN {X 0.008,Y -549.133,Z 575.168,A 0.000,B 0.000,C 90.000,E1 66.177} C_DIS
LIN {X 0.133,Y -542.754,Z 575.165,A 0.000,B 0.000,C 90.000,E1 65.741} C_DIS
LIN {X 0.216,Y -536.246,Z 575.163,A 0.000,B 0.000,C 90.000,E1 65.357} C_DIS
LIN {X -0.160,Y -529.565,Z 575.161,A 0.000,B 0.000,C 90.000,E1 65.049} C_DIS
LIN {X -0.155,Y -524.350,Z 575.160,A 0.000,B 0.000,C 90.000,E1 64.793} C_DIS
LIN {X -0.095,Y -514.088,Z 575.157,A 0.000,B 0.000,C 90.000,E1 64.332} C_DIS
LIN {X 0.153,Y -493.015,Z 575.153,A 0.000,B 0.000,C 90.000,E1 63.461} C_DIS
LIN {X -0.091,Y -475.840,Z 575.149,A 0.000,B 0.000,C 90.000,E1 62.794} C_DIS
LIN {X -0.294,Y -462.086,Z 575.146,A 0.000,B 0.000,C 90.000,E1 62.231} C_DIS
LIN {X -0.138,Y -455.486,Z 575.144,A 0.000,B 0.000,C 90.000,E1 61.897} C_DIS
LIN {X -0.179,Y -455.427,Z 575.144,A 0.000,B 0.000,C 90.000,E1 61.897} C_DIS
LIN {X -0.056,Y -445.802,Z 575.120,A 0.000,B 0.000,C 90.000,E1 57.533} C_DIS
LIN {X 0.003,Y -444.047,Z 575.114,A 0.000,B 0.000,C 90.000,E1 56.548} C_DIS
LIN {X -0.202,Y -436.428,Z 575.096,A 0.000,B 0.000,C 90.000,E1 53.336} C_DIS
LIN {X -0.057,Y -438.662,Z 575.085,A 0.000,B 0.000,C 90.000,E1 51.295} C_DIS
LIN {X 0.110,Y -440.819,Z 575.074,A 0.000,B 0.000,C 90.000,E1 49.299} C_DIS
LIN {X 0.278,Y -442.960,Z 575.063,A 0.000,B 0.000,C 90.000,E1 47.310} C_DIS
LIN {X -0.140,Y -444.681,Z 575.054,A 0.000,B 0.000,C 90.000,E1 45.729} C_DIS
LIN {X -0.203,Y -445.899,Z 575.047,A 0.000,B 0.000,C 90.000,E1 44.433} C_DIS
LIN {X 0.083,Y -446.687,Z 575.041,A 0.000,B 0.000,C 90.000,E1 43.419} C_DIS
LIN {X 0.053,Y -447.344,Z 575.036,A 0.000,B 0.000,C 90.000,E1 42.447} C_DIS
LIN {X 0.049,Y -448.067,Z 575.029,A 0.000,B 0.000,C 90.000,E1 41.148} C_DIS
LIN {X 0.052,Y -448.581,Z 575.021,A 0.000,B 0.000,C 90.000,E1 39.850} C_DIS
LIN {X -0.212,Y -448.869,Z 575.016,A 0.000,B 0.000,C 90.000,E1 38.910} C_DIS
LIN {X -0.131,Y -449.101,Z 575.009,A 0.000,B 0.000,C 90.000,E1 37.604} C_DIS
LIN {X 0.020,Y -449.130,Z 575.000,A 0.000,B 0.000,C 90.000,E1 35.964} C_DIS
LIN {X -0.135,Y -448.825,Z 574.989,A 0.000,B 0.000,C 90.000,E1 34.040} C_DIS
LIN {X -0.058,Y -448.490,Z 574.978,A 0.000,B 0.000,C 90.000,E1 32.084} C_DIS
LIN {X 0.016,Y -448.257,Z 574.967,A 0.000,B 0.000,C 90.000,E1 30.129} C_DIS
LIN {X 0.166,Y -448.084,Z 574.958,A 0.000,B 0.000,C 90.000,E1 28.487} C_DIS
LIN {X -0.033,Y -447.825,Z 574.948,A 0.000,B 0.000,C 90.000,E1 26.565} C_DIS
LIN {X 0.168,Y -447.635,Z 574.937,A 0.000,B 0.000,C 90.000,E1 24.591} C_DIS
LIN {X -0.160,Y -447.624,Z 574.930,A 0.000,B 0.000,C 90.000,E1 23.334} C_DIS
LIN {X -0.044,Y -447.712,Z 574.917,A 0.000,B 0.000,C 90.000,E1 21.046} C_DIS
LIN {X 0.034,Y -447.826,Z 574.906,A 0.000,B 0.000,C 90.000,E1 19.087} C_DIS
LIN {X -0.014,Y -448.134,Z 574.892,A 0.000,B 0.000,C 90.000,E1 16.496} C_DIS
LIN {X 0.087,Y -448.637,Z 574.881,A 0.000,B 0.000,C 90.000,E1 14.537} C_DIS
LIN {X -0.160,Y -449.469,Z 574.868,A 0.000,B 0.000,C 90.000,E1 12.299} C_DIS
LIN {X 0.010,Y -450.215,Z 574.859,A 0.000,B 0.000,C 90.000,E1 10.658} C_DIS
LIN {X 0.193,Y -451.741,Z 574.845,A 0.000,B 0.000,C 90.000,E1 8.049} C_DIS
LIN {X -0.137,Y -453.529,Z 574.831,A 0.000,B 0.000,C 90.000,E1 5.511} C_DIS
LIN {X -0.210,Y -455.485,Z 574.818,A 0.000,B 0.000,C 90.000,E1 3.269} C_DIS
LIN {X 0.007,Y -457.311,Z 574.807,A 0.000,B 0.000,C 90.000,E1 1.318} C_DIS
LIN {X 0.174,Y -459.047,Z 574.799,A 0.000,B 0.000,C 90.000,E1 359.771} C_DIS
LIN {X 0.154,Y -462.649,Z 574.783,A 0.000,B 0.000,C 90.000,E1 356.906} C_DIS
LIN {X 0.116,Y -465.366,Z 574.772,A 0.000,B 0.000,C 90.000,E1 355.008} C_DIS
LIN {X -0.050,Y -468.661,Z 574.760,A 0.000,B 0.000,C 90.000,E1 352.818} C_DIS
LIN {X 0.175,Y -471.519,Z 574.750,A 0.000,B 0.000,C 90.000,E1 350.905} C_DIS
LIN {X -0.174,Y -474.862,Z 574.737,A 0.000,B 0.000,C 90.000,E1 348.757} C_DIS
LIN {X 0.160,Y -478.768,Z 574.724,A 0.000,B 0.000,C 90.000,E1 346.228} C_DIS
LIN {X -0.178,Y -482.509,Z 574.712,A 0.000,B 0.000,C 90.000,E1 344.102} C_DIS
LIN {X -0.161,Y -486.538,Z 574.700,A 0.000,B 0.000,C 90.000,E1 341.945} C_DIS
LIN {X 0.249,Y -490.127,Z 574.689,A 0.000,B 0.000,C 90.000,E1 340.061} C_DIS
LIN {X -0.176,Y -493.594,Z 574.679,A 0.000,B 0.000,C 90.000,E1 338.284} C_DIS
LIN {X 0.005,Y -495.868,Z 574.673,A 0.000,B 0.000,C 90.000,E1 337.050} C_DIS
LIN {X 0.023,Y -498.552,Z 574.664,A 0.000,B 0.000,C 90.000,E1 335.537} C_DIS
LIN {X 0.154,Y -501.634,Z 574.654,A 0.000,B 0.000,C 90.000,E1 333.717} C_DIS
LIN {X 0.045,Y -504.042,Z 574.646,A 0.000,B 0.000,C 90.000,E1 332.231} C_DIS
LIN {X 0.224,Y -506.393,Z 574.638,A 0.000,B 0.000,C 90.000,E1 330.717} C_DIS
LIN {X -0.023,Y -509.797,Z 574.626,A 0.000,B 0.000,C 90.000,E1 328.663} C_DIS
LIN {X -0.273,Y -512.772,Z 574.616,A 0.000,B 0.000,C 90.000,E1 326.914} C_DIS
LIN {X 0.037,Y -516.338,Z 574.605,A 0.000,B 0.000,C 90.000,E1 324.815} C_DIS
LIN {X 0.139,Y -518.968,Z 574.596,A 0.000,B 0.000,C 90.000,E1 323.336} C_DIS
LIN {X 0.005,Y -523.836,Z 574.582,A 0.000,B 0.000,C 90.000,E1 320.723} C_DIS
LIN {X 0.084,Y -532.599,Z 574.559,A 0.000,B 0.000,C 90.000,E1 316.662} C_DIS
LIN {X -0.010,Y -534.754,Z 574.555,A 0.000,B 0.000,C 90.000,E1 315.810} C_DIS
LIN {X -0.074,Y -537.505,Z 574.550,A 0.000,B 0.000,C 90.000,E1 314.960} C_DIS
LIN {X -0.026,Y -538.400,Z 574.549,A 0.000,B 0.000,C 90.000,E1 314.757} C_DIS
LIN {X -0.240,Y -540.040,Z 574.546,A 0.000,B 0.000,C 90.000,E1 314.352} C_DIS
LIN {X 0.320,Y -542.375,Z 574.544,A 0.000,B 0.000,C 90.000,E1 313.866} C_DIS
LIN {X -0.162,Y -544.497,Z 574.542,A 0.000,B 0.000,C 90.000,E1 313.623} C_DIS
LIN {X 0.134,Y -548.433,Z 574.540,A 0.000,B 0.000,C 90.000,E1 313.137} C_DIS
LIN {X 0.081,Y -552.912,Z 574.537,A 0.000,B 0.000,C 90.000,E1 312.690} C_DIS
LIN {X -0.001,Y -557.850,Z 574.535,A 0.000,B 0.000,C 90.000,E1 312.285} C_DIS
LIN {X 0.120,Y -560.906,Z 574.534,A 0.000,B 0.000,C 90.000,E1 312.043} C_DIS
LIN {X -0.031,Y -566.821,Z 574.531,A 0.000,B 0.000,C 90.000,E1 311.595} C_DIS
LIN {X -0.255,Y -578.514,Z 574.526,A 0.000,B 0.000,C 90.000,E1 310.782} C_DIS
LIN {X -0.068,Y -591.882,Z 574.521,A 0.000,B 0.000,C 90.000,E1 309.806} C_DIS
LIN {X 0.121,Y -597.542,Z 574.519,A 0.000,B 0.000,C 90.000,E1 309.358} C_DIS
LIN {X -0.024,Y -601.719,Z 574.517,A 0.000,B 0.000,C 90.000,E1 309.036} C_DIS
LIN {X 0.230,Y -607.000,Z 574.514,A 0.000,B 0.000,C 90.000,E1 308.543} C_DIS
LIN {X 0.284,Y -610.853,Z 574.512,A 0.000,B 0.000,C 90.000,E1 308.177} C_DIS
LIN {X 0.083,Y -616.871,Z 574.509,A 0.000,B 0.000,C 90.000,E1 307.569} C_DIS
LIN {X 0.197,Y -623.892,Z 574.505,A 0.000,B 0.000,C 90.000,E1 306.790} C_DIS
LIN {X -0.004,Y -628.287,Z 574.502,A 0.000,B 0.000,C 90.000,E1 306.297} C_DIS
LIN {X 0.191,Y -634.419,Z 574.497,A 0.000,B 0.000,C 90.000,E1 305.518} C_DIS
LIN {X 0.070,Y -639.330,Z 574.494,A 0.000,B 0.000,C 90.000,E1 304.898} C_DIS
LIN {X 0.039,Y -643.844,Z 574.490,A 0.000,B 0.000,C 90.000,E1 304.278} C_DIS
LIN {X 0.193,Y -647.172,Z 574.488,A 0.000,B 0.000,C 90.000,E1 303.785} C_DIS
LIN {X 0.177,Y -651.000,Z 574.484,A 0.000,B 0.000,C 90.000,E1 303.166} C_DIS
LIN {X 0.148,Y -653.889,Z 574.482,A 0.000,B 0.000,C 90.000,E1 302.673} C_DIS
LIN {X 0.016,Y -657.564,Z 574.478,A 0.000,B 0.000,C 90.000,E1 301.957} C_DIS
LIN {X 0.137,Y -660.939,Z 574.474,A 0.000,B 0.000,C 90.000,E1 301.209} C_DIS
LIN {X -0.010,Y -666.230,Z 574.467,A 0.000,B 0.000,C 90.000,E1 300.001} C_DIS
LIN {X -0.296,Y -668.267,Z 574.464,A 0.000,B 0.000,C 90.000,E1 299.539} C_DIS
LIN {X 0.014,Y -670.032,Z 574.461,A 0.000,B 0.000,C 90.000,E1 299.027} C_DIS
LIN {X -0.412,Y -671.061,Z 574.460,A 0.000,B 0.000,C 90.000,E1 298.821} C_DIS
LIN {X -0.078,Y -672.649,Z 574.457,A 0.000,B 0.000,C 90.000,E1 298.309} C_DIS
LIN {X 0.094,Y -673.599,Z 574.456,A 0.000,B 0.000,C 90.000,E1 298.052} C_DIS
LIN {X -0.147,Y -675.098,Z 574.453,A 0.000,B 0.000,C 90.000,E1 297.590} C_DIS
LIN {X 0.034,Y -676.005,Z 574.452,A 0.000,B 0.000,C 90.000,E1 297.334} C_DIS
LIN {X -0.007,Y -678.324,Z 574.448,A 0.000,B 0.000,C 90.000,E1 296.616} C_DIS
LIN {X -0.229,Y -679.227,Z 574.445,A 0.000,B 0.000,C 90.000,E1 296.155} C_DIS
LIN {X -0.034,Y -679.337,Z 574.444,A 0.000,B 0.000,C 90.000,E1 295.899} C_DIS
LIN {X 0.067,Y -679.262,Z 574.441,A 0.000,B 0.000,C 90.000,E1 295.412} C_DIS
LIN {X 0.264,Y -678.572,Z 574.440,A 0.000,B 0.000,C 90.000,E1 295.155} C_DIS
LIN {X 0.037,Y -675.659,Z 574.437,A 0.000,B 0.000,C 90.000,E1 294.695} C_DIS
LIN {X -0.151,Y -674.759,Z 574.437,A 0.000,B 0.000,C 90.000,E1 294.591} C_DIS
LIN {X -0.058,Y -673.316,Z 574.436,A 0.000,B 0.000,C 90.000,E1 294.463} C_DIS
LIN {X -0.240,Y -669.517,Z 574.435,A 0.000,B 0.000,C 90.000,E1 294.259} C_DIS
LIN {X -0.183,Y -666.818,Z 574.434,A 0.000,B 0.000,C 90.000,E1 294.079} C_DIS
LIN {X 0.223,Y -664.729,Z 574.433,A 0.000,B 0.000,C 90.000,E1 293.951} C_DIS
LIN {X -0.250,Y -662.295,Z 574.433,A 0.000,B 0.000,C 90.000,E1 293.898} C_DIS
LIN {X 0.148,Y -656.867,Z 574.432,A 0.000,B 0.000,C 90.000,E1 293.695} C_DIS
LIN {X -0.201,Y -651.187,Z 574.431,A 0.000,B 0.000,C 90.000,E1 293.567} C_DIS
LIN {X 0.260,Y -618.901,Z 574.427,A 0.000,B 0.000,C 90.000,E1 292.770} C_DIS
LIN {X -0.005,Y -598.974,Z 574.423,A 0.000,B 0.000,C 90.000,E1 292.206} C_DIS
LIN {X -0.006,Y -578.314,Z 574.420,A 0.000,B 0.000,C 90.000,E1 291.535} C_DIS
LIN {X 0.184,Y -571.880,Z 574.418,A 0.000,B 0.000,C 90.000,E1 291.280} C_DIS
LIN {X 0.126,Y -566.528,Z 574.417,A 0.000,B 0.000,C 90.000,E1 291.046} C_DIS
LIN {X 0.079,Y -563.912,Z 574.416,A 0.000,B 0.000,C 90.000,E1 290.844} C_DIS
LIN {X 0.044,Y -563.892,Z 574.416,A 0.000,B 0.000,C 90.000,E1 290.844} C_DIS
LIN {X -0.126,Y -563.043,Z 574.415,A 0.000,B 0.000,C 90.000,E1 290.663} C_DIS
LIN {X -0.105,Y -562.718,Z 574.412,A 0.000,B 0.000,C 90.000,E1 290.248} C_DIS
LIN {X 0.052,Y -562.814,Z 574.405,A 0.000,B 0.000,C 90.000,E1 288.852} C_DIS
LIN {X 0.204,Y -562.494,Z 574.397,A 0.000,B 0.000,C 90.000,E1 287.457} C_DIS
LIN {X 0.173,Y -561.961,Z 574.389,A 0.000,B 0.000,C 90.000,E1 286.079} C_DIS
LIN {X -0.019,Y -561.248,Z 574.382,A 0.000,B 0.000,C 90.000,E1 284.717} C_DIS
LIN {X -0.223,Y -560.422,Z 574.374,A 0.000,B 0.000,C 90.000,E1 283.355} C_DIS
LIN {X -0.023,Y -559.651,Z 574.366,A 0.000,B 0.000,C 90.000,E1 281.951} C_DIS
LIN {X 0.164,Y -558.869,Z 574.359,A 0.000,B 0.000,C 90.000,E1 280.546} C_DIS
LIN {X 0.151,Y -557.465,Z 574.345,A 0.000,B 0.000,C 90.000,E1 278.049} C_DIS
LIN {X 0.117,Y -556.924,Z 574.337,A 0.000,B 0.000,C 90.000,E1 276.663} C_DIS
LIN {X -0.232,Y -556.090,Z 574.325,A 0.000,B 0.000,C 90.000,E1 274.473} C_DIS
LIN {X -0.135,Y -555.367,Z 574.312,A 0.000,B 0.000,C 90.000,E1 272.236} C_DIS
LIN {X -0.227,Y -554.771,Z 574.303,A 0.000,B 0.000,C 90.000,E1 270.573} C_DIS
LIN {X -0.275,Y -553.920,Z 574.292,A 0.000,B 0.000,C 90.000,E1 268.625} C_DIS
LIN {X 0.243,Y -553.104,Z 574.281,A 0.000,B 0.000,C 90.000,E1 266.617} C_DIS
LIN {X 0.030,Y -552.415,Z 574.274,A 0.000,B 0.000,C 90.000,E1 265.241} C_DIS
LIN {X -0.104,Y -551.621,Z 574.266,A 0.000,B 0.000,C 90.000,E1 263.856} C_DIS
LIN {X 0.198,Y -550.892,Z 574.260,A 0.000,B 0.000,C 90.000,E1 262.704} C_DIS
LIN {X -0.098,Y -550.140,Z 574.255,A 0.000,B 0.000,C 90.000,E1 261.894} C_DIS
LIN {X -0.185,Y -548.703,Z 574.247,A 0.000,B 0.000,C 90.000,E1 260.500} C_DIS
LIN {X -0.197,Y -547.038,Z 574.238,A 0.000,B 0.000,C 90.000,E1 258.814} C_DIS
LIN {X -0.146,Y -545.305,Z 574.228,A 0.000,B 0.000,C 90.000,E1 257.117} C_DIS
LIN {X -0.017,Y -543.508,Z 574.219,A 0.000,B 0.000,C 90.000,E1 255.408} C_DIS
LIN {X -0.161,Y -542.629,Z 574.214,A 0.000,B 0.000,C 90.000,E1 254.574} C_DIS
LIN {X -0.088,Y -541.289,Z 574.208,A 0.000,B 0.000,C 90.000,E1 253.433} C_DIS
LIN {X -0.193,Y -539.805,Z 574.202,A 0.000,B 0.000,C 90.000,E1 252.308} C_DIS
LIN {X 0.051,Y -537.804,Z 574.194,A 0.000,B 0.000,C 90.000,E1 250.859} C_DIS
LIN {X 0.224,Y -535.950,Z 574.187,A 0.000,B 0.000,C 90.000,E1 249.699} C_DIS
LIN {X -0.129,Y -533.929,Z 574.181,A 0.000,B 0.000,C 90.000,E1 248.592} C_DIS
LIN {X 0.186,Y -531.723,Z 574.175,A 0.000,B 0.000,C 90.000,E1 247.411} C_DIS
LIN {X -0.131,Y -528.080,Z 574.165,A 0.000,B 0.000,C 90.000,E1 245.717} C_DIS
LIN {X 0.090,Y -525.544,Z 574.159,A 0.000,B 0.000,C 90.000,E1 244.537} C_DIS
LIN {X 0.169,Y -522.228,Z 574.151,A 0.000,B 0.000,C 90.000,E1 243.076} C_DIS
LIN {X -0.090,Y -520.168,Z 574.146,A 0.000,B 0.000,C 90.000,E1 242.231} C_DIS
LIN {X -0.332,Y -516.481,Z 574.138,A 0.000,B 0.000,C 90.000,E1 240.795} C_DIS
LIN {X -0.035,Y -513.296,Z 574.131,A 0.000,B 0.000,C 90.000,E1 239.587} C_DIS
LIN {X -0.179,Y -507.500,Z 574.120,A 0.000,B 0.000,C 90.000,E1 237.533} C_DIS
LIN {X 0.030,Y -502.482,Z 574.110,A 0.000,B 0.000,C 90.000,E1 235.722} C_DIS
LIN {X 0.260,Y -498.221,Z 574.101,A 0.000,B 0.000,C 90.000,E1 234.196} C_DIS
LIN {X -0.134,Y -491.697,Z 574.088,A 0.000,B 0.000,C 90.000,E1 231.823} C_DIS
LIN {X 0.064,Y -486.095,Z 574.076,A 0.000,B 0.000,C 90.000,E1 229.666} C_DIS
LIN {X -0.259,Y -480.611,Z 574.064,A 0.000,B 0.000,C 90.000,E1 227.553} C_DIS
LIN {X 0.133,Y -476.022,Z 574.054,A 0.000,B 0.000,C 90.000,E1 225.648} C_DIS
LIN {X 0.167,Y -470.793,Z 574.042,A 0.000,B 0.000,C 90.000,E1 223.461} C_DIS
LIN {X 0.006,Y -466.473,Z 574.031,A 0.000,B 0.000,C 90.000,E1 221.595} C_DIS
LIN {X 0.196,Y -461.646,Z 574.019,A 0.000,B 0.000,C 90.000,E1 219.358} C_DIS
LIN {X -0.034,Y -456.844,Z 574.006,A 0.000,B 0.000,C 90.000,E1 217.156} C_DIS
LIN {X 0.250,Y -453.549,Z 573.998,A 0.000,B 0.000,C 90.000,E1 215.518} C_DIS
LIN {X 0.069,Y -448.348,Z 573.983,A 0.000,B 0.000,C 90.000,E1 212.959} C_DIS
LIN {X 0.183,Y -444.089,Z 573.971,A 0.000,B 0.000,C 90.000,E1 210.669} C_DIS
LIN {X -0.095,Y -440.539,Z 573.960,A 0.000,B 0.000,C 90.000,E1 208.743} C_DIS
LIN {X 0.243,Y -438.311,Z 573.952,A 0.000,B 0.000,C 90.000,E1 207.385} C_DIS
LIN {X -0.200,Y -434.851,Z 573.941,A 0.000,B 0.000,C 90.000,E1 205.463} C_DIS
LIN {X -0.149,Y -432.639,Z 573.934,A 0.000,B 0.000,C 90.000,E1 204.131} C_DIS
LIN {X -0.100,Y -429.953,Z 573.925,A 0.000,B 0.000,C 90.000,E1 202.461} C_DIS
LIN {X -0.098,Y -426.439,Z 573.912,A 0.000,B 0.000,C 90.000,E1 200.120} C_DIS
LIN {X -0.137,Y -423.585,Z 573.901,A 0.000,B 0.000,C 90.000,E1 198.109} C_DIS
LIN {X 0.125,Y -420.028,Z 573.886,A 0.000,B 0.000,C 90.000,E1 195.371} C_DIS
LIN {X -0.088,Y -417.937,Z 573.876,A 0.000,B 0.000,C 90.000,E1 193.703} C_DIS
LIN {X -0.187,Y -415.985,Z 573.869,A 0.000,B 0.000,C 90.000,E1 192.355} C_DIS
LIN {X -0.108,Y -411.801,Z 573.851,A 0.000,B 0.000,C 90.000,E1 189.265} C_DIS
LIN {X 0.048,Y -409.035,Z 573.838,A 0.000,B 0.000,C 90.000,E1 186.834} C_DIS
LIN {X 0.058,Y -406.739,Z 573.827,A 0.000,B 0.000,C 90.000,E1 184.759} C_DIS
LIN {X -0.164,Y -403.299,Z 573.807,A 0.000,B 0.000,C 90.000,E1 181.318} C_DIS
LIN {X -0.013,Y -401.544,Z 573.794,A 0.000,B 0.000,C 90.000,E1 178.854} C_DIS
LIN {X 0.112,Y -400.126,Z 573.780,A 0.000,B 0.000,C 90.000,E1 176.388} C_DIS
LIN {X 0.178,Y -399.075,Z 573.763,A 0.000,B 0.000,C 90.000,E1 173.223} C_DIS
LIN {X -0.003,Y -398.695,Z 573.749,A 0.000,B 0.000,C 90.000,E1 170.792} C_DIS
LIN {X -0.118,Y -398.637,Z 573.737,A 0.000,B 0.000,C 90.000,E1 168.701} C_DIS
LIN {X 0.035,Y -399.084,Z 573.720,A 0.000,B 0.000,C 90.000,E1 165.519} C_DIS
LIN {X -0.131,Y -399.776,Z 573.706,A 0.000,B 0.000,C 90.000,E1 163.087} C_DIS
LIN {X 0.074,Y -400.659,Z 573.692,A 0.000,B 0.000,C 90.000,E1 160.604} C_DIS
LIN {X -0.162,Y -401.646,Z 573.681,A 0.000,B 0.000,C 90.000,E1 158.539} C_DIS
LIN {X -0.091,Y -402.692,Z 573.669,A 0.000,B 0.000,C 90.000,E1 156.433} C_DIS
LIN {X -0.032,Y -403.802,Z 573.657,A 0.000,B 0.000,C 90.000,E1 154.332} C_DIS
LIN {X 0.060,Y -404.927,Z 573.646,A 0.000,B 0.000,C 90.000,E1 152.231} C_DIS
LIN {X 0.028,Y -405.679,Z 573.638,A 0.000,B 0.000,C 90.000,E1 150.845} C_DIS
LIN {X -0.077,Y -406.447,Z 573.628,A 0.000,B 0.000,C 90.000,E1 149.125} C_DIS
LIN {X 0.040,Y -407.036,Z 573.619,A 0.000,B 0.000,C 90.000,E1 147.375} C_DIS
LIN {X -0.181,Y -407.498,Z 573.609,A 0.000,B 0.000,C 90.000,E1 145.674} C_DIS
LIN {X 0.065,Y -407.884,Z 573.600,A 0.000,B 0.000,C 90.000,E1 143.909} C_DIS
LIN {X -0.008,Y -408.180,Z 573.590,A 0.000,B 0.000,C 90.000,E1 142.190} C_DIS
LIN {X 0.010,Y -408.446,Z 573.578,A 0.000,B 0.000,C 90.000,E1 140.114} C_DIS
LIN {X -0.123,Y -408.693,Z 573.569,A 0.000,B 0.000,C 90.000,E1 138.405} C_DIS
LIN {X 0.131,Y -408.817,Z 573.557,A 0.000,B 0.000,C 90.000,E1 136.296} C_DIS
LIN {X 0.228,Y -409.100,Z 573.544,A 0.000,B 0.000,C 90.000,E1 133.866} C_DIS
LIN {X 0.069,Y -409.319,Z 573.534,A 0.000,B 0.000,C 90.000,E1 132.162} C_DIS
LIN {X 0.068,Y -409.355,Z 573.527,A 0.000,B 0.000,C 90.000,E1 130.782} C_DIS
LIN {X -0.092,Y -409.312,Z 573.521,A 0.000,B 0.000,C 90.000,E1 129.769} C_DIS
LIN {X -0.205,Y -409.155,Z 573.515,A 0.000,B 0.000,C 90.000,E1 128.749} C_DIS
LIN {X 0.035,Y -409.060,Z 573.512,A 0.000,B 0.000,C 90.000,E1 128.177} C_DIS
LIN {X 0.012,Y -415.548,Z 573.500,A 0.000,B 0.000,C 90.000,E1 125.964} C_DIS
LIN {X 0.095,Y -425.939,Z 573.477,A 0.000,B 0.000,C 90.000,E1 121.878} C_DIS
LIN {X 0.049,Y -430.946,Z 573.468,A 0.000,B 0.000,C 90.000,E1 120.207} C_DIS
LIN {X 0.060,Y -434.316,Z 573.460,A 0.000,B 0.000,C 90.000,E1 118.743} C_DIS
LIN {X 0.021,Y -434.353,Z 573.460,A 0.000,B 0.000,C 90.000,E1 118.743} C_DIS
LIN {X -0.193,Y -449.247,Z 573.456,A 0.000,B 0.000,C 90.000,E1 118.103} C_DIS
LIN {X -0.072,Y -468.116,Z 573.451,A 0.000,B 0.000,C 90.000,E1 117.206} C_DIS
LIN {X 0.017,Y -476.545,Z 573.449,A 0.000,B 0.000,C 90.000,E1 116.796} C_DIS
LIN {X 0.215,Y -490.092,Z 573.445,A 0.000,B 0.000,C 90.000,E1 116.104} C_DIS
LIN {X 0.060,Y -499.917,Z 573.442,A 0.000,B 0.000,C 90.000,E1 115.591} C_DIS
LIN {X -0.029,Y -511.226,Z 573.439,A 0.000,B 0.000,C 90.000,E1 114.951} C_DIS
LIN {X -0.232,Y -517.702,Z 573.437,A 0.000,B 0.000,C 90.000,E1 114.591} C_DIS
LIN {X -0.126,Y -528.774,Z 573.433,A 0.000,B 0.000,C 90.000,E1 113.875} C_DIS
LIN {X -0.133,Y -539.386,Z 573.428,A 0.000,B 0.000,C 90.000,E1 113.131} C_DIS
LIN {X -0.102,Y -546.693,Z 573.425,A 0.000,B 0.000,C 90.000,E1 112.567} C_DIS
LIN {X -0.084,Y -549.689,Z 573.424,A 0.000,B 0.000,C 90.000,E1 112.333} C_DIS
LIN {X 0.073,Y -555.088,Z 573.421,A 0.000,B 0.000,C 90.000,E1 111.844} C_DIS
LIN {X -0.106,Y -560.344,Z 573.419,A 0.000,B 0.000,C 90.000,E1 111.354} C_DIS
LIN {X -0.163,Y -563.806,Z 573.416,A 0.000,B 0.000,C 90.000,E1 110.972} C_DIS
LIN {X 0.259,Y -565.175,Z 573.416,A 0.000,B 0.000,C 90.000,E1 110.791} C_DIS
LIN {X 0.232,Y -570.992,Z 573.412,A 0.000,B 0.000,C 90.000,E1 110.066} C_DIS
LIN {X 0.041,Y -572.785,Z 573.410,A 0.000,B 0.000,C 90.000,E1 109.812} C_DIS
LIN {X 0.032,Y -575.350,Z 573.408,A 0.000,B 0.000,C 90.000,E1 109.450} C_DIS
LIN {X -0.052,Y -579.640,Z 573.404,A 0.000,B 0.000,C 90.000,E1 108.779} C_DIS
LIN {X 0.196,Y -584.204,Z 573.400,A 0.000,B 0.000,C 90.000,E1 107.946} C_DIS
LIN {X 0.080,Y -588.269,Z 573.395,A 0.000,B 0.000,C 90.000,E1 107.166} C_DIS
LIN {X 0.106,Y -591.525,Z 573.392,A 0.000,B 0.000,C 90.000,E1 106.496} C_DIS
LIN {X -0.015,Y -594.568,Z 573.388,A 0.000,B 0.000,C 90.000,E1 105.843} C_DIS
LIN {X -0.180,Y -597.990,Z 573.384,A 0.000,B 0.000,C 90.000,E1 105.064} C_DIS
LIN {X -0.184,Y -600.195,Z 573.381,A 0.000,B 0.000,C 90.000,E1 104.537} C_DIS
LIN {X 0.318,Y -605.261,Z 573.373,A 0.000,B 0.000,C 90.000,E1 103.175} C_DIS
LIN {X -0.205,Y -611.164,Z 573.365,A 0.000,B 0.000,C 90.000,E1 101.658} C_DIS
LIN {X -0.004,Y -615.084,Z 573.359,A 0.000,B 0.000,C 90.000,E1 100.602} C_DIS
LIN {X -0.103,Y -619.769,Z 573.352,A 0.000,B 0.000,C 90.000,E1 99.321} C_DIS
LIN {X -0.289,Y -622.525,Z 573.347,A 0.000,B 0.000,C 90.000,E1 98.568} C_DIS
LIN {X 0.260,Y -627.033,Z 573.340,A 0.000,B 0.000,C 90.000,E1 97.239} C_DIS
LIN {X 0.261,Y -631.170,Z 573.333,A 0.000,B 0.000,C 90.000,E1 95.967} C_DIS
LIN {X -0.157,Y -634.129,Z 573.328,A 0.000,B 0.000,C 90.000,E1 94.992} C_DIS
LIN {X -0.269,Y -636.125,Z 573.323,A 0.000,B 0.000,C 90.000,E1 94.245} C_DIS
LIN {X 0.273,Y -637.860,Z 573.319,A 0.000,B 0.000,C 90.000,E1 93.440} C_DIS
LIN {X 0.195,Y -639.432,Z 573.315,A 0.000,B 0.000,C 90.000,E1 92.694} C_DIS
LIN {X 0.104,Y -640.789,Z 573.311,A 0.000,B 0.000,C 90.000,E1 91.949} C_DIS
LIN {X 0.047,Y -641.916,Z 573.307,A 0.000,B 0.000,C 90.000,E1 91.203} C_DIS
LIN {X -0.249,Y -643.069,Z 573.301,A 0.000,B 0.000,C 90.000,E1 90.229} C_DIS
LIN {X 0.113,Y -643.698,Z 573.296,A 0.000,B 0.000,C 90.000,E1 89.198} C_DIS
LIN {X 0.295,Y -643.823,Z 573.293,A 0.000,B 0.000,C 90.000,E1 88.682} C_DIS
LIN {X 0.269,Y -643.854,Z 573.289,A 0.000,B 0.000,C 90.000,E1 87.936} C_DIS
LIN {X -0.014,Y -643.423,Z 573.283,A 0.000,B 0.000,C 90.000,E1 86.963} C_DIS
LIN {X -0.040,Y -642.923,Z 573.279,A 0.000,B 0.000,C 90.000,E1 86.216} C_DIS
LIN {X -0.310,Y -641.825,Z 573.273,A 0.000,B 0.000,C 90.000,E1 85.241} C_DIS
LIN {X -0.291,Y -640.888,Z 573.269,A 0.000,B 0.000,C 90.000,E1 84.489} C_DIS
LIN {X 0.298,Y -639.741,Z 573.265,A 0.000,B 0.000,C 90.000,E1 83.685} C_DIS
LIN {X 0.045,Y -637.909,Z 573.260,A 0.000,B 0.000,C 90.000,E1 82.704} C_DIS
LIN {X 0.224,Y -636.846,Z 573.257,A 0.000,B 0.000,C 90.000,E1 82.186} C_DIS
LIN {X -0.264,Y -633.813,Z 573.250,A 0.000,B 0.000,C 90.000,E1 80.971} C_DIS
LIN {X 0.118,Y -631.085,Z 573.244,A 0.000,B 0.000,C 90.000,E1 79.926} C_DIS
LIN {X -0.360,Y -627.356,Z 573.237,A 0.000,B 0.000,C 90.000,E1 78.701} C_DIS
LIN {X 0.053,Y -624.099,Z 573.231,A 0.000,B 0.000,C 90.000,E1 77.645} C_DIS
LIN {X 0.241,Y -622.378,Z 573.229,A 0.000,B 0.000,C 90.000,E1 77.117} C_DIS
LIN {X -0.022,Y -618.563,Z 573.223,A 0.000,B 0.000,C 90.000,E1 76.117} C_DIS
LIN {X -0.180,Y -614.331,Z 573.217,A 0.000,B 0.000,C 90.000,E1 75.102} C_DIS
LIN {X -0.304,Y -610.896,Z 573.213,A 0.000,B 0.000,C 90.000,E1 74.338} C_DIS
LIN {X -0.046,Y -608.420,Z 573.210,A 0.000,B 0.000,C 90.000,E1 73.795} C_DIS
LIN {X -0.027,Y -605.156,Z 573.206,A 0.000,B 0.000,C 90.000,E1 73.142} C_DIS
LIN {X -0.039,Y -601.736,Z 573.203,A 0.000,B 0.000,C 90.000,E1 72.489} C_DIS
LIN {X 0.048,Y -597.204,Z 573.198,A 0.000,B 0.000,C 90.000,E1 71.692} C_DIS
LIN {X 0.234,Y -592.334,Z 573.194,A 0.000,B 0.000,C 90.000,E1 70.913} C_DIS
LIN {X -0.197,Y -588.717,Z 573.191,A 0.000,B 0.000,C 90.000,E1 70.423} C_DIS
LIN {X 0.273,Y -584.127,Z 573.188,A 0.000,B 0.000,C 90.000,E1 69.752} C_DIS
LIN {X 0.108,Y -579.042,Z 573.184,A 0.000,B 0.000,C 90.000,E1 69.135} C_DIS
LIN {X -0.078,Y -573.313,Z 573.181,A 0.000,B 0.000,C 90.000,E1 68.518} C_DIS
LIN {X 0.283,Y -568.463,Z 573.178,A 0.000,B 0.000,C 90.000,E1 67.975} C_DIS
LIN {X -0.155,Y -563.482,Z 573.175,A 0.000,B 0.000,C 90.000,E1 67.539} C_DIS
LIN {X 0.207,Y -558.415,Z 573.173,A 0.000,B 0.000,C 90.000,E1 67.050} C_DIS
LIN {X 0.083,Y -552.726,Z 573.170,A 0.000,B 0.000,C 90.000,E1 66.613} C_DIS
LIN {X 0.117,Y -548.463,Z 573.168,A 0.000,B 0.000,C 90.000,E1 66.305} C_DIS
LIN {X -0.205,Y -541.968,Z 573.166,A 0.000,B 0.000,C 90.000,E1 65.921} C_DIS
LIN {X -0.053,Y -536.845,Z 573.165,A 0.000,B 0.000,C 90.000,E1 65.613} C_DIS
LIN {X -0.090,Y -528.289,Z 573.162,A 0.000,B 0.000,C 90.000,E1 65.177} C_DIS
LIN {X 0.275,Y -524.965,Z 573.161,A 0.000,B 0.000,C 90.000,E1 64.973} C_DIS
LIN {X 0.182,Y -517.723,Z 573.159,A 0.000,B 0.000,C 90.000,E1 64.665} C_DIS
LIN {X -0.116,Y -510.591,Z 573.158,A 0.000,B 0.000,C 90.000,E1 64.409} C_DIS
LIN {X 0.073,Y -489.912,Z 573.153,A 0.000,B 0.000,C 90.000,E1 63.563} C_DIS
LIN {X 0.193,Y -476.070,Z 573.150,A 0.000,B 0.000,C 90.000,E1 62.999} C_DIS
LIN {X 0.097,Y -459.101,Z 573.146,A 0.000,B 0.000,C 90.000,E1 62.281} C_DIS
LIN {X -0.101,Y -455.940,Z 573.145,A 0.000,B 0.000,C 90.000,E1 62.153} C_DIS
LIN {X -0.143,Y -455.857,Z 573.145,A 0.000,B 0.000,C 90.000,E1 62.153} C_DIS
LIN {X 0.143,Y -454.893,Z 573.143,A 0.000,B 0.000,C 90.000,E1 61.641} C_DIS
LIN {X 0.042,Y -445.678,Z 573.119,A 0.000,B 0.000,C 90.000,E1 57.454} C_DIS
LIN {X -0.143,Y -443.922,Z 573.114,A 0.000,B 0.000,C 90.000,E1 56.501} C_DIS
LIN {X -0.052,Y -436.813,Z 573.097,A 0.000,B 0.000,C 90.000,E1 53.497} C_DIS
LIN {X -0.172,Y -438.654,Z 573.088,A 0.000,B 0.000,C 90.000,E1 51.904} C_DIS
LIN {X -0.009,Y -440.847,Z 573.077,A 0.000,B 0.000,C 90.000,E1 49.908} C_DIS
LIN {X 0.189,Y -442.708,Z 573.068,A 0.000,B 0.000,C 90.000,E1 48.243} C_DIS
LIN {X 0.090,Y -444.496,Z 573.059,A 0.000,B 0.000,C 90.000,E1 46.620} C_DIS
LIN {X 0.008,Y -446.191,Z 573.050,A 0.000,B 0.000,C 90.000,E1 45.000} C_DIS
LIN {X -0.033,Y -447.295,Z 573.043,A 0.000,B 0.000,C 90.000,E1 43.704} C_DIS
LIN {X -0.040,Y -448.204,Z 573.036,A 0.000,B 0.000,C 90.000,E1 42.405} C_DIS
LIN {X 0.272,Y -448.938,Z 573.028,A 0.000,B 0.000,C 90.000,E1 41.067} C_DIS
LIN {X 0.000,Y -449.414,Z 573.021,A 0.000,B 0.000,C 90.000,E1 39.806} C_DIS
LIN {X -0.262,Y -449.730,Z 573.014,A 0.000,B 0.000,C 90.000,E1 38.543} C_DIS
LIN {X 0.125,Y -449.889,Z 573.009,A 0.000,B 0.000,C 90.000,E1 37.523} C_DIS
LIN {X -0.077,Y -449.816,Z 573.000,A 0.000,B 0.000,C 90.000,E1 35.931} C_DIS
LIN {X -0.185,Y -449.526,Z 572.991,A 0.000,B 0.000,C 90.000,E1 34.326} C_DIS
LIN {X 0.230,Y -449.097,Z 572.978,A 0.000,B 0.000,C 90.000,E1 32.005} C_DIS
LIN {X 0.088,Y -448.828,Z 572.967,A 0.000,B 0.000,C 90.000,E1 30.079} C_DIS
LIN {X -0.214,Y -448.676,Z 572.960,A 0.000,B 0.000,C 90.000,E1 28.821} C_DIS
LIN {X -0.059,Y -448.435,Z 572.951,A 0.000,B 0.000,C 90.000,E1 27.180} C_DIS
LIN {X 0.016,Y -448.148,Z 572.938,A 0.000,B 0.000,C 90.000,E1 24.899} C_DIS
LIN {X 0.155,Y -448.050,Z 572.929,A 0.000,B 0.000,C 90.000,E1 23.259} C_DIS
LIN {X -0.058,Y -448.059,Z 572.920,A 0.000,B 0.000,C 90.000,E1 21.663} C_DIS
LIN {X 0.035,Y -448.150,Z 572.910,A 0.000,B 0.000,C 90.000,E1 19.704} C_DIS
LIN {X -0.122,Y -448.436,Z 572.893,A 0.000,B 0.000,C 90.000,E1 16.804} C_DIS
LIN {X -0.147,Y -448.935,Z 572.881,A 0.000,B 0.000,C 90.000,E1 14.537} C_DIS
LIN {X 0.053,Y -449.749,Z 572.868,A 0.000,B 0.000,C 90.000,E1 12.243} C_DIS
LIN {X 0.230,Y -450.477,Z 572.859,A 0.000,B 0.000,C 90.000,E1 10.602} C_DIS
LIN {X -0.022,Y -451.969,Z 572.845,A 0.000,B 0.000,C 90.000,E1 8.049} C_DIS
LIN {X 0.105,Y -453.744,Z 572.830,A 0.000,B 0.000,C 90.000,E1 5.454} C_DIS
LIN {X 0.041,Y -455.682,Z 572.818,A 0.000,B 0.000,C 90.000,E1 3.212} C_DIS
LIN {X 0.184,Y -458.216,Z 572.804,A 0.000,B 0.000,C 90.000,E1 0.630} C_DIS
LIN {X -0.213,Y -461.070,Z 572.790,A 0.000,B 0.000,C 90.000,E1 358.224} C_DIS
LIN {X -0.117,Y -464.115,Z 572.778,A 0.000,B 0.000,C 90.000,E1 355.988} C_DIS
LIN {X 0.128,Y -466.378,Z 572.769,A 0.000,B 0.000,C 90.000,E1 354.375} C_DIS
LIN {X 0.236,Y -469.233,Z 572.758,A 0.000,B 0.000,C 90.000,E1 352.470} C_DIS
LIN {X -0.066,Y -472.077,Z 572.748,A 0.000,B 0.000,C 90.000,E1 350.622} C_DIS
LIN {X 0.141,Y -475.415,Z 572.736,A 0.000,B 0.000,C 90.000,E1 348.409} C_DIS
LIN {X 0.023,Y -479.316,Z 572.722,A 0.000,B 0.000,C 90.000,E1 345.936} C_DIS
LIN {X 0.145,Y -483.694,Z 572.708,A 0.000,B 0.000,C 90.000,E1 343.449} C_DIS
LIN {X -0.118,Y -487.768,Z 572.696,A 0.000,B 0.000,C 90.000,E1 341.329} C_DIS
LIN {X 0.299,Y -490.751,Z 572.688,A 0.000,B 0.000,C 90.000,E1 339.752} C_DIS
LIN {X -0.155,Y -493.636,Z 572.679,A 0.000,B 0.000,C 90.000,E1 338.284} C_DIS
LIN {X 0.078,Y -496.470,Z 572.671,A 0.000,B 0.000,C 90.000,E1 336.741} C_DIS
LIN {X 0.046,Y -498.627,Z 572.664,A 0.000,B 0.000,C 90.000,E1 335.537} C_DIS
LIN {X 0.019,Y -502.208,Z 572.652,A 0.000,B 0.000,C 90.000,E1 333.435} C_DIS
LIN {X -0.069,Y -504.606,Z 572.644,A 0.000,B 0.000,C 90.000,E1 331.948} C_DIS
LIN {X -0.119,Y -506.966,Z 572.636,A 0.000,B 0.000,C 90.000,E1 330.461} C_DIS
LIN {X 0.008,Y -509.918,Z 572.626,A 0.000,B 0.000,C 90.000,E1 328.663} C_DIS
LIN {X -0.238,Y -512.919,Z 572.616,A 0.000,B 0.000,C 90.000,E1 326.914} C_DIS
LIN {X 0.076,Y -516.473,Z 572.605,A 0.000,B 0.000,C 90.000,E1 324.815} C_DIS
LIN {X 0.181,Y -519.095,Z 572.596,A 0.000,B 0.000,C 90.000,E1 323.336} C_DIS
LIN {X 0.095,Y -523.372,Z 572.583,A 0.000,B 0.000,C 90.000,E1 321.009} C_DIS
LIN {X -0.251,Y -527.416,Z 572.572,A 0.000,B 0.000,C 90.000,E1 319.013} C_DIS
LIN {X 0.138,Y -532.633,Z 572.559,A 0.000,B 0.000,C 90.000,E1 316.662} C_DIS
LIN {X 0.019,Y -535.535,Z 572.553,A 0.000,B 0.000,C 90.000,E1 315.526} C_DIS
LIN {X -0.035,Y -537.188,Z 572.550,A 0.000,B 0.000,C 90.000,E1 314.960} C_DIS
LIN {X 0.308,Y -539.173,Z 572.547,A 0.000,B 0.000,C 90.000,E1 314.352} C_DIS
LIN {X -0.088,Y -540.584,Z 572.545,A 0.000,B 0.000,C 90.000,E1 314.109} C_DIS
LIN {X 0.287,Y -541.707,Z 572.543,A 0.000,B 0.000,C 90.000,E1 313.785} C_DIS
LIN {X -0.102,Y -543.324,Z 572.542,A 0.000,B 0.000,C 90.000,E1 313.542} C_DIS
LIN {X -0.092,Y -545.205,Z 572.540,A 0.000,B 0.000,C 90.000,E1 313.257} C_DIS
LIN {X -0.017,Y -549.103,Z 572.538,A 0.000,B 0.000,C 90.000,E1 312.771} C_DIS
LIN {X -0.118,Y -552.371,Z 572.536,A 0.000,B 0.000,C 90.000,E1 312.447} C_DIS
LIN {X -0.226,Y -560.557,Z 572.532,A 0.000,B 0.000,C 90.000,E1 311.757} C_DIS
LIN {X 0.347,Y -567.864,Z 572.529,A 0.000,B 0.000,C 90.000,E1 311.148} C_DIS
LIN {X 0.008,Y -581.383,Z 572.523,A 0.000,B 0.000,C 90.000,E1 310.216} C_DIS
LIN {X -0.036,Y -591.641,Z 572.519,A 0.000,B 0.000,C 90.000,E1 309.483} C_DIS
LIN {X 0.026,Y -596.002,Z 572.518,A 0.000,B 0.000,C 90.000,E1 309.152} C_DIS
LIN {X -0.081,Y -600.168,Z 572.516,A 0.000,B 0.000,C 90.000,E1 308.830} C_DIS
LIN {X -0.136,Y -605.311,Z 572.513,A 0.000,B 0.000,C 90.000,E1 308.382} C_DIS
LIN {X -0.037,Y -610.337,Z 572.511,A 0.000,B 0.000,C 90.000,E1 307.890} C_DIS
LIN {X -0.153,Y -614.165,Z 572.508,A 0.000,B 0.000,C 90.000,E1 307.523} C_DIS
LIN {X 0.306,Y -622.445,Z 572.503,A 0.000,B 0.000,C 90.000,E1 306.583} C_DIS
LIN {X -0.075,Y -629.993,Z 572.498,A 0.000,B 0.000,C 90.000,E1 305.724} C_DIS
LIN {X 0.134,Y -636.036,Z 572.494,A 0.000,B 0.000,C 90.000,E1 304.945} C_DIS
LIN {X 0.043,Y -641.844,Z 572.490,A 0.000,B 0.000,C 90.000,E1 304.199} C_DIS
LIN {X -0.016,Y -646.133,Z 572.487,A 0.000,B 0.000,C 90.000,E1 303.579} C_DIS
LIN {X -0.076,Y -649.358,Z 572.484,A 0.000,B 0.000,C 90.000,E1 303.086} C_DIS
LIN {X -0.076,Y -652.929,Z 572.480,A 0.000,B 0.000,C 90.000,E1 302.467} C_DIS
LIN {X -0.398,Y -656.117,Z 572.477,A 0.000,B 0.000,C 90.000,E1 301.878} C_DIS
LIN {X 0.158,Y -658.484,Z 572.474,A 0.000,B 0.000,C 90.000,E1 301.337} C_DIS
LIN {X -0.031,Y -663.775,Z 572.467,A 0.000,B 0.000,C 90.000,E1 300.129} C_DIS
LIN {X -0.189,Y -666.773,Z 572.463,A 0.000,B 0.000,C 90.000,E1 299.411} C_DIS
LIN {X -0.318,Y -669.552,Z 572.459,A 0.000,B 0.000,C 90.000,E1 298.693} C_DIS
LIN {X -0.249,Y -672.895,Z 572.454,A 0.000,B 0.000,C 90.000,E1 297.719} C_DIS
LIN {X -0.320,Y -675.376,Z 572.450,A 0.000,B 0.000,C 90.000,E1 297.001} C_DIS
LIN {X 0.047,Y -676.835,Z 572.447,A 0.000,B 0.000,C 90.000,E1 296.488} C_DIS
LIN {X 0.234,Y -677.392,Z 572.446,A 0.000,B 0.000,C 90.000,E1 296.232} C_DIS
LIN {X -0.186,Y -677.690,Z 572.445,A 0.000,B 0.000,C 90.000,E1 296.027} C_DIS
LIN {X -0.097,Y -677.709,Z 572.442,A 0.000,B 0.000,C 90.000,E1 295.540} C_DIS
LIN {X 0.096,Y -677.337,Z 572.441,A 0.000,B 0.000,C 90.000,E1 295.283} C_DIS
LIN {X 0.192,Y -676.816,Z 572.440,A 0.000,B 0.000,C 90.000,E1 295.155} C_DIS
LIN {X -0.047,Y -673.902,Z 572.437,A 0.000,B 0.000,C 90.000,E1 294.695} C_DIS
LIN {X -0.236,Y -672.731,Z 572.437,A 0.000,B 0.000,C 90.000,E1 294.591} C_DIS
LIN {X -0.059,Y -668.753,Z 572.435,A 0.000,B 0.000,C 90.000,E1 294.335} C_DIS
LIN {X -0.058,Y -666.824,Z 572.434,A 0.000,B 0.000,C 90.000,E1 294.155} C_DIS
LIN {X 0.043,Y -664.683,Z 572.434,A 0.000,B 0.000,C 90.000,E1 294.027} C_DIS
LIN {X 0.239,Y -658.488,Z 572.432,A 0.000,B 0.000,C 90.000,E1 293.770} C_DIS
LIN {X -0.271,Y -652.562,Z 572.431,A 0.000,B 0.000,C 90.000,E1 293.643} C_DIS
LIN {X 0.138,Y -647.038,Z 572.430,A 0.000,B 0.000,C 90.000,E1 293.462} C_DIS
LIN {X 0.074,Y -630.755,Z 572.428,A 0.000,B 0.000,C 90.000,E1 293.078} C_DIS
LIN {X 0.139,Y -620.258,Z 572.427,A 0.000,B 0.000,C 90.000,E1 292.823} C_DIS
LIN {X -0.056,Y -600.265,Z 572.424,A 0.000,B 0.000,C 90.000,E1 292.259} C_DIS
LIN {X -0.009,Y -579.666,Z 572.420,A 0.000,B 0.000,C 90.000,E1 291.589} C_DIS
LIN {X 0.088,Y -573.432,Z 572.419,A 0.000,B 0.000,C 90.000,E1 291.354} C_DIS
LIN {X -0.271,Y -566.992,Z 572.417,A 0.000,B 0.000,C 90.000,E1 291.099} C_DIS
LIN {X 0.024,Y -564.225,Z 572.416,A 0.000,B 0.000,C 90.000,E1 290.844} C_DIS
LIN {X -0.013,Y -564.208,Z 572.416,A 0.000,B 0.000,C 90.000,E1 290.844} C_DIS
LIN {X -0.121,Y -563.706,Z 572.415,A 0.000,B 0.000,C 90.000,E1 290.737} C_DIS
LIN {X -0.013,Y -563.429,Z 572.415,A 0.000,B 0.000,C 90.000,E1 290.610} C_DIS
LIN {X -0.307,Y -563.185,Z 572.412,A 0.000,B 0.000,C 90.000,E1 290.248} C_DIS
LIN {X 0.255,Y -563.272,Z 572.406,A 0.000,B 0.000,C 90.000,E1 289.087} C_DIS
LIN {X 0.097,Y -563.117,Z 572.400,A 0.000,B 0.000,C 90.000,E1 288.000} C_DIS
LIN {X -0.065,Y -562.748,Z 572.394,A 0.000,B 0.000,C 90.000,E1 286.913} C_DIS
LIN {X 0.145,Y -562.276,Z 572.388,A 0.000,B 0.000,C 90.000,E1 285.788} C_DIS
LIN {X -0.036,Y -561.550,Z 572.380,A 0.000,B 0.000,C 90.000,E1 284.426} C_DIS
LIN {X 0.070,Y -560.422,Z 572.369,A 0.000,B 0.000,C 90.000,E1 282.479} C_DIS
LIN {X -0.127,Y -559.466,Z 572.360,A 0.000,B 0.000,C 90.000,E1 280.838} C_DIS
LIN {X 0.239,Y -558.325,Z 572.349,A 0.000,B 0.000,C 90.000,E1 278.859} C_DIS
LIN {X -0.069,Y -557.487,Z 572.339,A 0.000,B 0.000,C 90.000,E1 276.947} C_DIS
LIN {X 0.024,Y -556.713,Z 572.328,A 0.000,B 0.000,C 90.000,E1 274.992} C_DIS
LIN {X -0.082,Y -556.218,Z 572.320,A 0.000,B 0.000,C 90.000,E1 273.612} C_DIS
LIN {X -0.232,Y -555.802,Z 572.312,A 0.000,B 0.000,C 90.000,E1 272.236} C_DIS
LIN {X 0.241,Y -555.174,Z 572.303,A 0.000,B 0.000,C 90.000,E1 270.516} C_DIS
LIN {X 0.203,Y -554.323,Z 572.292,A 0.000,B 0.000,C 90.000,E1 268.568} C_DIS
LIN {X 0.081,Y -553.619,Z 572.283,A 0.000,B 0.000,C 90.000,E1 266.906} C_DIS
